gfCNCPoint1[18036] = {X 7.8608, Y 36.7035, Z -1.3333, A 0.000, B 0.000, C 0.000 }
gfCNCPoint1[18037] = {X 8.3776, Y 37.1520, Z -1.3333, A 0.000, B 0.000, C 0.000 }
gfCNCPoint1[18038] = {X 9.1826, Y 37.5595, Z -1.3333, A 0.000, B 0.000, C 0.000 }
gfCNCPoint1[18039] = {X 10.0390, Y 37.8436, Z -1.3333, A 0.000, B 0.000, C 0.000 }
gfCNCPoint1[18040] = {X 11.3458, Y 38.0858, Z -1.3333, A 0.000, B 0.000, C 0.000 }
gfCNCPoint1[18041] = {X 12.6726, Y 38.1626, Z -1.3333, A 0.000, B 0.000, C 0.000 }
gfCNCPoint1[18042] = {X 13.9985, Y 38.0726, Z -1.3333, A 0.000, B 0.000, C 0.000 }
gfCNCPoint1[18043] = {X 15.3028, Y 37.8174, Z -1.3333, A 0.000, B 0.000, C 0.000 }
gfCNCPoint1[18044] = {X 16.5649, Y 37.4009, Z -1.3333, A 0.000, B 0.000, C 0.000 }
gfCNCPoint1[18045] = {X 17.9591, Y 36.7477, Z -1.3333, A 0.000, B 0.000, C 0.000 }
gfCNCPoint1[18046] = {X 19.2706, Y 35.9412, Z -1.3333, A 0.000, B 0.000, C 0.000 }
gfCNCPoint1[18047] = {X 19.3492, Y 35.2028, Z -1.3333, A 0.000, B 0.000, C 0.000 }
gfCNCPoint1[18048] = {X 19.5579, Y 34.4902, Z -1.3333, A 0.000, B 0.000, C 0.000 }
gfCNCPoint1[18049] = {X 19.8900, Y 33.8261, Z -1.3333, A 0.000, B 0.000, C 0.000 }
gfCNCPoint1[18050] = {X 18.0017, Y 34.1716, Z -1.3333, A 0.000, B 0.000, C 0.000 }
gfCNCPoint1[18051] = {X 16.0932, Y 34.3789, Z -1.3333, A 0.000, B 0.000, C 0.000 }
gfCNCPoint1[18052] = {X 15.3691, Y 34.4315, Z -1.3333, A 0.000, B 0.000, C 0.000 }
gfCNCPoint1[18053] = {X 14.6448, Y 34.4821, Z -1.3333, A 0.000, B 0.000, C 0.000 }
gfCNCPoint1[18054] = {X 10.6931, Y 35.1018, Z -1.3333, A 0.000, B 0.000, C 0.000 }
gfCNCPoint1[18055] = {X 18.6386, Y 34.4782, Z -1.3333, A 0.000, B 0.000, C 0.000 }
gfCNCPoint1[18056] = {X 14.6393, Y 34.4023, Z -1.3333, A 0.000, B 0.000, C 0.000 }
gfCNCPoint1[18057] = {X 12.2464, Y 34.5545, Z -1.3333, A 0.000, B 0.000, C 0.000 }
gfCNCPoint1[18058] = {X 9.8522, Y 34.6839, Z -1.3333, A 0.000, B 0.000, C 0.000 }
gfCNCPoint1[18059] = {X 8.6234, Y 34.7897, Z -1.3333, A 0.000, B 0.000, C 0.000 }
gfCNCPoint1[18060] = {X 7.4164, Y 35.0431, Z -1.3333, A 0.000, B 0.000, C 0.000 }
gfCNCPoint1[18061] = {X 7.3529, Y 35.2331, Z -1.3333, A 0.000, B 0.000, C 0.000 }
gfCNCPoint1[18062] = {X 7.3309, Y 35.4323, Z -1.3333, A 0.000, B 0.000, C 0.000 }
gfCNCPoint1[18063] = {X 7.3977, Y 35.9629, Z -1.3333, A 0.000, B 0.000, C 0.000 }
gfCNCPoint1[18064] = {X 7.5977, Y 36.4590, Z -1.3333, A 0.000, B 0.000, C 0.000 }
gfCNCPoint1[18065] = {X 7.9176, Y 36.8876, Z -1.3333, A 0.000, B 0.000, C 0.000 }
gfCNCPoint1[18066] = {X 8.3362, Y 37.2205, Z -1.3333, A 0.000, B 0.000, C 0.000 }
gfCNCPoint1[18067] = {X 9.1519, Y 37.6334, Z -1.3333, A 0.000, B 0.000, C 0.000 }
gfCNCPoint1[18068] = {X 10.0195, Y 37.9212, Z -1.3333, A 0.000, B 0.000, C 0.000 }
gfCNCPoint1[18069] = {X 11.3362, Y 38.1652, Z -1.3333, A 0.000, B 0.000, C 0.000 }
gfCNCPoint1[18070] = {X 12.6730, Y 38.2425, Z -1.3333, A 0.000, B 0.000, C 0.000 }
gfCNCPoint1[18071] = {X 14.0089, Y 38.1519, Z -1.3333, A 0.000, B 0.000, C 0.000 }
gfCNCPoint1[18072] = {X 15.3231, Y 37.8948, Z -1.3333, A 0.000, B 0.000, C 0.000 }
gfCNCPoint1[18073] = {X 16.5947, Y 37.4752, Z -1.3333, A 0.000, B 0.000, C 0.000 }
gfCNCPoint1[18074] = {X 18.0152, Y 36.8083, Z -1.3333, A 0.000, B 0.000, C 0.000 }
gfCNCPoint1[18075] = {X 19.3501, Y 35.9832, Z -1.3333, A 0.000, B 0.000, C 0.000 }
gfCNCPoint1[18076] = {X 19.4352, Y 35.1814, Z -1.3333, A 0.000, B 0.000, C 0.000 }
gfCNCPoint1[18077] = {X 19.6764, Y 34.4119, Z -1.3333, A 0.000, B 0.000, C 0.000 }
gfCNCPoint1[18078] = {X 20.0642, Y 33.7049, Z -1.3333, A 0.000, B 0.000, C 0.000 }
gfCNCPoint1[18079] = {X 18.0872, Y 34.0781, Z -1.3333, A 0.000, B 0.000, C 0.000 }
gfCNCPoint1[18080] = {X 16.0874, Y 34.2991, Z -1.3333, A 0.000, B 0.000, C 0.000 }
gfCNCPoint1[18081] = {X 15.3634, Y 34.3517, Z -1.3333, A 0.000, B 0.000, C 0.000 }
gfCNCPoint1[18082] = {X 14.6393, Y 34.4023, Z -1.3333, A 0.000, B 0.000, C 0.000 }
gfCNCPoint1[18083] = {X 10.6876, Y 35.0220, Z -1.3333, A 0.000, B 0.000, C 0.000 }
gfCNCPoint1[18084] = {X 14.7703, Y 36.3178, Z -1.3333, A 0.000, B 0.000, C 0.000 }
gfCNCPoint1[18085] = {X 14.6338, Y 34.3225, Z -1.3333, A 0.000, B 0.000, C 0.000 }
gfCNCPoint1[18086] = {X 12.2422, Y 34.4746, Z -1.3333, A 0.000, B 0.000, C 0.000 }
gfCNCPoint1[18087] = {X 9.8492, Y 34.6040, Z -1.3333, A 0.000, B 0.000, C 0.000 }
gfCNCPoint1[18088] = {X 8.5932, Y 34.7133, Z -1.3333, A 0.000, B 0.000, C 0.000 }
gfCNCPoint1[18089] = {X 7.3600, Y 34.9757, Z -1.3333, A 0.000, B 0.000, C 0.000 }
gfCNCPoint1[18090] = {X 7.2790, Y 35.1975, Z -1.3333, A 0.000, B 0.000, C 0.000 }
gfCNCPoint1[18091] = {X 7.2509, Y 35.4320, Z -1.3333, A 0.000, B 0.000, C 0.000 }
gfCNCPoint1[18092] = {X 7.3203, Y 35.9830, Z -1.3333, A 0.000, B 0.000, C 0.000 }
gfCNCPoint1[18093] = {X 7.5280, Y 36.4982, Z -1.3333, A 0.000, B 0.000, C 0.000 }
gfCNCPoint1[18094] = {X 7.8602, Y 36.9433, Z -1.3333, A 0.000, B 0.000, C 0.000 }
gfCNCPoint1[18095] = {X 8.2949, Y 37.2890, Z -1.3333, A 0.000, B 0.000, C 0.000 }
gfCNCPoint1[18096] = {X 9.1211, Y 37.7073, Z -1.3333, A 0.000, B 0.000, C 0.000 }
gfCNCPoint1[18097] = {X 10.0001, Y 37.9988, Z -1.3333, A 0.000, B 0.000, C 0.000 }
gfCNCPoint1[18098] = {X 11.3265, Y 38.2446, Z -1.3333, A 0.000, B 0.000, C 0.000 }
gfCNCPoint1[18099] = {X 12.6734, Y 38.3225, Z -1.3333, A 0.000, B 0.000, C 0.000 }
gfCNCPoint1[18100] = {X 14.0194, Y 38.2312, Z -1.3333, A 0.000, B 0.000, C 0.000 }
gfCNCPoint1[18101] = {X 15.3433, Y 37.9722, Z -1.3333, A 0.000, B 0.000, C 0.000 }
gfCNCPoint1[18102] = {X 16.6244, Y 37.5494, Z -1.3333, A 0.000, B 0.000, C 0.000 }
gfCNCPoint1[18103] = {X 18.0716, Y 36.8688, Z -1.3333, A 0.000, B 0.000, C 0.000 }
gfCNCPoint1[18104] = {X 19.4300, Y 36.0248, Z -1.3333, A 0.000, B 0.000, C 0.000 }
gfCNCPoint1[18105] = {X 19.5226, Y 35.1553, Z -1.3333, A 0.000, B 0.000, C 0.000 }
gfCNCPoint1[18106] = {X 19.8019, Y 34.3266, Z -1.3333, A 0.000, B 0.000, C 0.000 }
gfCNCPoint1[18107] = {X 20.2547, Y 33.5784, Z -1.3333, A 0.000, B 0.000, C 0.000 }
gfCNCPoint1[18108] = {X 18.1810, Y 33.9830, Z -1.3333, A 0.000, B 0.000, C 0.000 }
gfCNCPoint1[18109] = {X 16.0816, Y 34.2193, Z -1.3333, A 0.000, B 0.000, C 0.000 }
gfCNCPoint1[18110] = {X 15.3578, Y 34.2719, Z -1.3333, A 0.000, B 0.000, C 0.000 }
gfCNCPoint1[18111] = {X 14.6338, Y 34.3225, Z -1.3333, A 0.000, B 0.000, C 0.000 }
gfCNCPoint1[18112] = {X 14.7703, Y 36.3178, Z -1.3333, A 0.000, B 0.000, C 0.000 }
gfCNCPoint1[18113] = {X 14.7703, Y 36.3178, Z 1.6667, A 0.000, B 0.000, C 0.000 }
gfCNCPoint1[18114] = {X 14.7703, Y 36.3178, Z 11.0000, A 0.000, B 0.000, C 0.000 }
gfCNCPoint1[18115] = {X 15.0706, Y 19.4899, Z 11.0000, A 0.000, B 0.000, C 0.000 }
gfCNCPoint1[18116] = {X 15.0706, Y 19.4899, Z 2.5000, A 0.000, B 0.000, C 0.000 }
gfCNCPoint1[18117] = {X 14.5039, Y 19.3617, Z 2.3443, A 0.000, B 0.000, C 0.000 }
gfCNCPoint1[18118] = {X 13.3045, Y 19.2481, Z 2.0215, A 0.000, B 0.000, C 0.000 }
gfCNCPoint1[18119] = {X 12.0998, Y 19.2655, Z 1.6987, A 0.000, B 0.000, C 0.000 }
gfCNCPoint1[18120] = {X 11.2937, Y 19.3811, Z 1.4805, A 0.000, B 0.000, C 0.000 }
gfCNCPoint1[18121] = {X 10.6070, Y 19.4891, Z 1.2942, A 0.000, B 0.000, C 0.000 }
gfCNCPoint1[18122] = {X 9.8986, Y 19.6124, Z 1.1015, A 0.000, B 0.000, C 0.000 }
gfCNCPoint1[18123] = {X 8.6156, Y 20.0582, Z 0.7376, A 0.000, B 0.000, C 0.000 }
gfCNCPoint1[18124] = {X 7.9834, Y 20.4007, Z 0.5449, A 0.000, B 0.000, C 0.000 }
gfCNCPoint1[18125] = {X 7.9275, Y 20.9124, Z 0.4070, A 0.000, B 0.000, C 0.000 }
gfCNCPoint1[18126] = {X 7.4464, Y 22.1372, Z 0.0544, A 0.000, B 0.000, C 0.000 }
gfCNCPoint1[18127] = {X 7.1391, Y 22.5500, Z -0.0835, A 0.000, B 0.000, C 0.000 }
gfCNCPoint1[18128] = {X 8.7346, Y 22.3449, Z -0.5145, A 0.000, B 0.000, C 0.000 }
gfCNCPoint1[18129] = {X 9.6130, Y 22.2741, Z -0.7506, A 0.000, B 0.000, C 0.000 }
gfCNCPoint1[18130] = {X 11.2207, Y 22.2213, Z -1.1817, A 0.000, B 0.000, C 0.000 }
gfCNCPoint1[18131] = {X 11.5036, Y 22.2116, Z -1.2575, A 0.000, B 0.000, C 0.000 }
gfCNCPoint1[18132] = {X 11.7864, Y 22.2003, Z -1.3333, A 0.000, B 0.000, C 0.000 }
gfCNCPoint1[18133] = {X 14.1145, Y 22.0807, Z -1.3333, A 0.000, B 0.000, C 0.000 }
gfCNCPoint1[18134] = {X 16.4392, Y 21.9079, Z -1.3333, A 0.000, B 0.000, C 0.000 }
gfCNCPoint1[18135] = {X 17.0540, Y 21.8327, Z -1.3333, A 0.000, B 0.000, C 0.000 }
gfCNCPoint1[18136] = {X 17.6536, Y 21.6779, Z -1.3333, A 0.000, B 0.000, C 0.000 }
gfCNCPoint1[18137] = {X 17.6759, Y 21.2173, Z -1.3333, A 0.000, B 0.000, C 0.000 }
gfCNCPoint1[18138] = {X 17.5258, Y 20.7814, Z -1.3333, A 0.000, B 0.000, C 0.000 }
gfCNCPoint1[18139] = {X 17.2248, Y 20.4321, Z -1.3333, A 0.000, B 0.000, C 0.000 }
gfCNCPoint1[18140] = {X 16.3055, Y 19.8916, Z -1.3333, A 0.000, B 0.000, C 0.000 }
gfCNCPoint1[18141] = {X 15.2982, Y 19.5414, Z -1.3333, A 0.000, B 0.000, C 0.000 }
gfCNCPoint1[18142] = {X 13.9732, Y 19.3253, Z -1.3333, A 0.000, B 0.000, C 0.000 }
gfCNCPoint1[18143] = {X 12.6317, Y 19.2716, Z -1.3333, A 0.000, B 0.000, C 0.000 }
gfCNCPoint1[18144] = {X 11.2937, Y 19.3811, Z -1.3333, A 0.000, B 0.000, C 0.000 }
gfCNCPoint1[18145] = {X 10.6070, Y 19.4891, Z -1.3333, A 0.000, B 0.000, C 0.000 }
gfCNCPoint1[18146] = {X 9.2582, Y 19.8383, Z -1.3333, A 0.000, B 0.000, C 0.000 }
gfCNCPoint1[18147] = {X 7.9834, Y 20.4007, Z -1.3333, A 0.000, B 0.000, C 0.000 }
gfCNCPoint1[18148] = {X 7.8310, Y 21.1635, Z -1.3333, A 0.000, B 0.000, C 0.000 }
gfCNCPoint1[18149] = {X 7.5466, Y 21.8875, Z -1.3333, A 0.000, B 0.000, C 0.000 }
gfCNCPoint1[18150] = {X 7.1391, Y 22.5500, Z -1.3333, A 0.000, B 0.000, C 0.000 }
gfCNCPoint1[18151] = {X 9.1760, Y 22.3372, Z -1.3333, A 0.000, B 0.000, C 0.000 }
gfCNCPoint1[18152] = {X 11.2207, Y 22.2213, Z -1.3333, A 0.000, B 0.000, C 0.000 }
gfCNCPoint1[18153] = {X 11.5036, Y 22.2112, Z -1.3333, A 0.000, B 0.000, C 0.000 }
gfCNCPoint1[18154] = {X 11.7864, Y 22.2003, Z -1.3333, A 0.000, B 0.000, C 0.000 }
gfCNCPoint1[18155] = {X 7.7941, Y 22.0908, Z -1.3333, A 0.000, B 0.000, C 0.000 }
gfCNCPoint1[18156] = {X 11.7896, Y 22.2802, Z -1.3333, A 0.000, B 0.000, C 0.000 }
gfCNCPoint1[18157] = {X 14.1160, Y 22.1607, Z -1.3333, A 0.000, B 0.000, C 0.000 }
gfCNCPoint1[18158] = {X 16.4391, Y 21.9880, Z -1.3333, A 0.000, B 0.000, C 0.000 }
gfCNCPoint1[18159] = {X 17.0880, Y 21.9077, Z -1.3333, A 0.000, B 0.000, C 0.000 }
gfCNCPoint1[18160] = {X 17.7200, Y 21.7400, Z -1.3333, A 0.000, B 0.000, C 0.000 }
gfCNCPoint1[18161] = {X 17.7589, Y 21.2351, Z -1.3333, A 0.000, B 0.000, C 0.000 }
gfCNCPoint1[18162] = {X 17.6020, Y 20.7536, Z -1.3333, A 0.000, B 0.000, C 0.000 }
gfCNCPoint1[18163] = {X 17.2732, Y 20.3684, Z -1.3333, A 0.000, B 0.000, C 0.000 }
gfCNCPoint1[18164] = {X 16.3395, Y 19.8192, Z -1.3333, A 0.000, B 0.000, C 0.000 }
gfCNCPoint1[18165] = {X 15.3164, Y 19.4635, Z -1.3333, A 0.000, B 0.000, C 0.000 }
gfCNCPoint1[18166] = {X 13.9814, Y 19.2457, Z -1.3333, A 0.000, B 0.000, C 0.000 }
gfCNCPoint1[18167] = {X 12.6299, Y 19.1916, Z -1.3333, A 0.000, B 0.000, C 0.000 }
gfCNCPoint1[18168] = {X 11.2818, Y 19.3020, Z -1.3333, A 0.000, B 0.000, C 0.000 }
gfCNCPoint1[18169] = {X 10.5939, Y 19.4102, Z -1.3333, A 0.000, B 0.000, C 0.000 }
gfCNCPoint1[18170] = {X 9.2123, Y 19.7696, Z -1.3333, A 0.000, B 0.000, C 0.000 }
gfCNCPoint1[18171] = {X 7.9082, Y 20.3506, Z -1.3333, A 0.000, B 0.000, C 0.000 }
gfCNCPoint1[18172] = {X 7.7437, Y 21.1760, Z -1.3333, A 0.000, B 0.000, C 0.000 }
gfCNCPoint1[18173] = {X 7.4223, Y 21.9539, Z -1.3333, A 0.000, B 0.000, C 0.000 }
gfCNCPoint1[18174] = {X 6.9562, Y 22.6547, Z -1.3333, A 0.000, B 0.000, C 0.000 }
gfCNCPoint1[18175] = {X 9.0854, Y 22.4248, Z -1.3333, A 0.000, B 0.000, C 0.000 }
gfCNCPoint1[18176] = {X 11.2234, Y 22.3012, Z -1.3333, A 0.000, B 0.000, C 0.000 }
gfCNCPoint1[18177] = {X 11.5065, Y 22.2911, Z -1.3333, A 0.000, B 0.000, C 0.000 }
gfCNCPoint1[18178] = {X 11.7896, Y 22.2802, Z -1.3333, A 0.000, B 0.000, C 0.000 }
gfCNCPoint1[18179] = {X 15.7573, Y 21.7730, Z -1.3333, A 0.000, B 0.000, C 0.000 }
gfCNCPoint1[18180] = {X 7.7973, Y 22.1707, Z -1.3333, A 0.000, B 0.000, C 0.000 }
gfCNCPoint1[18181] = {X 11.7928, Y 22.3601, Z -1.3333, A 0.000, B 0.000, C 0.000 }
gfCNCPoint1[18182] = {X 14.1204, Y 22.2406, Z -1.3333, A 0.000, B 0.000, C 0.000 }
gfCNCPoint1[18183] = {X 16.4447, Y 22.0679, Z -1.3333, A 0.000, B 0.000, C 0.000 }
gfCNCPoint1[18184] = {X 17.1242, Y 21.9821, Z -1.3333, A 0.000, B 0.000, C 0.000 }
gfCNCPoint1[18185] = {X 17.7850, Y 21.8022, Z -1.3333, A 0.000, B 0.000, C 0.000 }
gfCNCPoint1[18186] = {X 17.8413, Y 21.2532, Z -1.3333, A 0.000, B 0.000, C 0.000 }
gfCNCPoint1[18187] = {X 17.6781, Y 20.7259, Z -1.3333, A 0.000, B 0.000, C 0.000 }
gfCNCPoint1[18188] = {X 17.3216, Y 20.3046, Z -1.3333, A 0.000, B 0.000, C 0.000 }
gfCNCPoint1[18189] = {X 16.3735, Y 19.7468, Z -1.3333, A 0.000, B 0.000, C 0.000 }
gfCNCPoint1[18190] = {X 15.3345, Y 19.3856, Z -1.3333, A 0.000, B 0.000, C 0.000 }
gfCNCPoint1[18191] = {X 13.9896, Y 19.1661, Z -1.3333, A 0.000, B 0.000, C 0.000 }
gfCNCPoint1[18192] = {X 12.6280, Y 19.1116, Z -1.3333, A 0.000, B 0.000, C 0.000 }
gfCNCPoint1[18193] = {X 11.2699, Y 19.2229, Z -1.3333, A 0.000, B 0.000, C 0.000 }
gfCNCPoint1[18194] = {X 10.5809, Y 19.3312, Z -1.3333, A 0.000, B 0.000, C 0.000 }
gfCNCPoint1[18195] = {X 9.6302, Y 19.5517, Z -1.3333, A 0.000, B 0.000, C 0.000 }
gfCNCPoint1[18196] = {X 8.7100, Y 19.8764, Z -1.3333, A 0.000, B 0.000, C 0.000 }
gfCNCPoint1[18197] = {X 7.8316, Y 20.3015, Z -1.3333, A 0.000, B 0.000, C 0.000 }
gfCNCPoint1[18198] = {X 7.8286, Y 20.3427, Z -1.3333, A 0.000, B 0.000, C 0.000 }
gfCNCPoint1[18199] = {X 7.6465, Y 21.2191, Z -1.3333, A 0.000, B 0.000, C 0.000 }
gfCNCPoint1[18200] = {X 7.2844, Y 22.0378, Z -1.3333, A 0.000, B 0.000, C 0.000 }
gfCNCPoint1[18201] = {X 6.7585, Y 22.7622, Z -1.3333, A 0.000, B 0.000, C 0.000 }
gfCNCPoint1[18202] = {X 8.9873, Y 22.5134, Z -1.3333, A 0.000, B 0.000, C 0.000 }
gfCNCPoint1[18203] = {X 11.2261, Y 22.3812, Z -1.3333, A 0.000, B 0.000, C 0.000 }
gfCNCPoint1[18204] = {X 11.5095, Y 22.3711, Z -1.3333, A 0.000, B 0.000, C 0.000 }
gfCNCPoint1[18205] = {X 11.7928, Y 22.3601, Z -1.3333, A 0.000, B 0.000, C 0.000 }
gfCNCPoint1[18206] = {X 15.7605, Y 21.8529, Z -1.3333, A 0.000, B 0.000, C 0.000 }
gfCNCPoint1[18207] = {X 7.8005, Y 22.2506, Z -1.3333, A 0.000, B 0.000, C 0.000 }
gfCNCPoint1[18208] = {X 11.7960, Y 22.4401, Z -1.3333, A 0.000, B 0.000, C 0.000 }
gfCNCPoint1[18209] = {X 14.1248, Y 22.3205, Z -1.3333, A 0.000, B 0.000, C 0.000 }
gfCNCPoint1[18210] = {X 16.4504, Y 22.1477, Z -1.3333, A 0.000, B 0.000, C 0.000 }
gfCNCPoint1[18211] = {X 17.1598, Y 22.0566, Z -1.3333, A 0.000, B 0.000, C 0.000 }
gfCNCPoint1[18212] = {X 17.8488, Y 21.8646, Z -1.3333, A 0.000, B 0.000, C 0.000 }
gfCNCPoint1[18213] = {X 17.9277, Y 21.4220, Z -1.3333, A 0.000, B 0.000, C 0.000 }
gfCNCPoint1[18214] = {X 17.8684, Y 20.9763, Z -1.3333, A 0.000, B 0.000, C 0.000 }
gfCNCPoint1[18215] = {X 17.6764, Y 20.5698, Z -1.3333, A 0.000, B 0.000, C 0.000 }
gfCNCPoint1[18216] = {X 17.3699, Y 20.2409, Z -1.3333, A 0.000, B 0.000, C 0.000 }
gfCNCPoint1[18217] = {X 16.4075, Y 19.6744, Z -1.3333, A 0.000, B 0.000, C 0.000 }
gfCNCPoint1[18218] = {X 15.3527, Y 19.3077, Z -1.3333, A 0.000, B 0.000, C 0.000 }
gfCNCPoint1[18219] = {X 13.9979, Y 19.0866, Z -1.3333, A 0.000, B 0.000, C 0.000 }
gfCNCPoint1[18220] = {X 12.6262, Y 19.0317, Z -1.3333, A 0.000, B 0.000, C 0.000 }
gfCNCPoint1[18221] = {X 11.2580, Y 19.1438, Z -1.3333, A 0.000, B 0.000, C 0.000 }
gfCNCPoint1[18222] = {X 10.5678, Y 19.2523, Z -1.3333, A 0.000, B 0.000, C 0.000 }
gfCNCPoint1[18223] = {X 9.5943, Y 19.4788, Z -1.3333, A 0.000, B 0.000, C 0.000 }
gfCNCPoint1[18224] = {X 8.6526, Y 19.8137, Z -1.3333, A 0.000, B 0.000, C 0.000 }
gfCNCPoint1[18225] = {X 7.7547, Y 20.2528, Z -1.3333, A 0.000, B 0.000, C 0.000 }
gfCNCPoint1[18226] = {X 7.7493, Y 20.3317, Z -1.3333, A 0.000, B 0.000, C 0.000 }
gfCNCPoint1[18227] = {X 7.5471, Y 21.2648, Z -1.3333, A 0.000, B 0.000, C 0.000 }
gfCNCPoint1[18228] = {X 7.1375, Y 22.1272, Z -1.3333, A 0.000, B 0.000, C 0.000 }
gfCNCPoint1[18229] = {X 6.5421, Y 22.8735, Z -1.3333, A 0.000, B 0.000, C 0.000 }
gfCNCPoint1[18230] = {X 8.8798, Y 22.6030, Z -1.3333, A 0.000, B 0.000, C 0.000 }
gfCNCPoint1[18231] = {X 11.2288, Y 22.4611, Z -1.3333, A 0.000, B 0.000, C 0.000 }
gfCNCPoint1[18232] = {X 11.5124, Y 22.4510, Z -1.3333, A 0.000, B 0.000, C 0.000 }
gfCNCPoint1[18233] = {X 11.7960, Y 22.4401, Z -1.3333, A 0.000, B 0.000, C 0.000 }
gfCNCPoint1[18234] = {X 15.7637, Y 21.9328, Z -1.3333, A 0.000, B 0.000, C 0.000 }
gfCNCPoint1[18235] = {X 7.8037, Y 22.3306, Z -1.3333, A 0.000, B 0.000, C 0.000 }
gfCNCPoint1[18236] = {X 11.7992, Y 22.5200, Z -1.3333, A 0.000, B 0.000, C 0.000 }
gfCNCPoint1[18237] = {X 14.1293, Y 22.4004, Z -1.3333, A 0.000, B 0.000, C 0.000 }
gfCNCPoint1[18238] = {X 16.4560, Y 22.2275, Z -1.3333, A 0.000, B 0.000, C 0.000 }
gfCNCPoint1[18239] = {X 17.1948, Y 22.1310, Z -1.3333, A 0.000, B 0.000, C 0.000 }
gfCNCPoint1[18240] = {X 17.9114, Y 21.9269, Z -1.3333, A 0.000, B 0.000, C 0.000 }
gfCNCPoint1[18241] = {X 18.0068, Y 21.4523, Z -1.3333, A 0.000, B 0.000, C 0.000 }
gfCNCPoint1[18242] = {X 17.9503, Y 20.9716, Z -1.3333, A 0.000, B 0.000, C 0.000 }
gfCNCPoint1[18243] = {X 17.7474, Y 20.5320, Z -1.3333, A 0.000, B 0.000, C 0.000 }
gfCNCPoint1[18244] = {X 17.4182, Y 20.1771, Z -1.3333, A 0.000, B 0.000, C 0.000 }
gfCNCPoint1[18245] = {X 16.4415, Y 19.6020, Z -1.3333, A 0.000, B 0.000, C 0.000 }
gfCNCPoint1[18246] = {X 15.3709, Y 19.2298, Z -1.3333, A 0.000, B 0.000, C 0.000 }
gfCNCPoint1[18247] = {X 14.0061, Y 19.0070, Z -1.3333, A 0.000, B 0.000, C 0.000 }
gfCNCPoint1[18248] = {X 12.6243, Y 18.9517, Z -1.3333, A 0.000, B 0.000, C 0.000 }
gfCNCPoint1[18249] = {X 11.2461, Y 19.0647, Z -1.3333, A 0.000, B 0.000, C 0.000 }
gfCNCPoint1[18250] = {X 10.5548, Y 19.1734, Z -1.3333, A 0.000, B 0.000, C 0.000 }
gfCNCPoint1[18251] = {X 9.5584, Y 19.4060, Z -1.3333, A 0.000, B 0.000, C 0.000 }
gfCNCPoint1[18252] = {X 8.5952, Y 19.7511, Z -1.3333, A 0.000, B 0.000, C 0.000 }
gfCNCPoint1[18253] = {X 7.6779, Y 20.2043, Z -1.3333, A 0.000, B 0.000, C 0.000 }
gfCNCPoint1[18254] = {X 7.6696, Y 20.3250, Z -1.3333, A 0.000, B 0.000, C 0.000 }
gfCNCPoint1[18255] = {X 7.5229, Y 21.0766, Z -1.3333, A 0.000, B 0.000, C 0.000 }
gfCNCPoint1[18256] = {X 7.2384, Y 21.7876, Z -1.3333, A 0.000, B 0.000, C 0.000 }
gfCNCPoint1[18257] = {X 6.8261, Y 22.4329, Z -1.3333, A 0.000, B 0.000, C 0.000 }
gfCNCPoint1[18258] = {X 6.3004, Y 22.9898, Z -1.3333, A 0.000, B 0.000, C 0.000 }
gfCNCPoint1[18259] = {X 8.7595, Y 22.6941, Z -1.3333, A 0.000, B 0.000, C 0.000 }
gfCNCPoint1[18260] = {X 11.2315, Y 22.5411, Z -1.3333, A 0.000, B 0.000, C 0.000 }
gfCNCPoint1[18261] = {X 11.5153, Y 22.5310, Z -1.3333, A 0.000, B 0.000, C 0.000 }
gfCNCPoint1[18262] = {X 11.7992, Y 22.5200, Z -1.3333, A 0.000, B 0.000, C 0.000 }
gfCNCPoint1[18263] = {X 15.7669, Y 22.0128, Z -1.3333, A 0.000, B 0.000, C 0.000 }
gfCNCPoint1[18264] = {X 11.7273, Y 22.6029, Z -1.3333, A 0.000, B 0.000, C 0.000 }
gfCNCPoint1[18265] = {X 11.8024, Y 22.6000, Z -1.3333, A 0.000, B 0.000, C 0.000 }
gfCNCPoint1[18266] = {X 14.1337, Y 22.4802, Z -1.3333, A 0.000, B 0.000, C 0.000 }
gfCNCPoint1[18267] = {X 16.4617, Y 22.3073, Z -1.3333, A 0.000, B 0.000, C 0.000 }
gfCNCPoint1[18268] = {X 17.2294, Y 22.2056, Z -1.3333, A 0.000, B 0.000, C 0.000 }
gfCNCPoint1[18269] = {X 17.9731, Y 21.9894, Z -1.3333, A 0.000, B 0.000, C 0.000 }
gfCNCPoint1[18270] = {X 18.0854, Y 21.4830, Z -1.3333, A 0.000, B 0.000, C 0.000 }
gfCNCPoint1[18271] = {X 18.0320, Y 20.9671, Z -1.3333, A 0.000, B 0.000, C 0.000 }
gfCNCPoint1[18272] = {X 17.8185, Y 20.4944, Z -1.3333, A 0.000, B 0.000, C 0.000 }
gfCNCPoint1[18273] = {X 17.4665, Y 20.1133, Z -1.3333, A 0.000, B 0.000, C 0.000 }
gfCNCPoint1[18274] = {X 16.4755, Y 19.5295, Z -1.3333, A 0.000, B 0.000, C 0.000 }
gfCNCPoint1[18275] = {X 15.3891, Y 19.1519, Z -1.3333, A 0.000, B 0.000, C 0.000 }
gfCNCPoint1[18276] = {X 14.0143, Y 18.9274, Z -1.3333, A 0.000, B 0.000, C 0.000 }
gfCNCPoint1[18277] = {X 12.6225, Y 18.8717, Z -1.3333, A 0.000, B 0.000, C 0.000 }
gfCNCPoint1[18278] = {X 11.2342, Y 18.9856, Z -1.3333, A 0.000, B 0.000, C 0.000 }
gfCNCPoint1[18279] = {X 10.5417, Y 19.0944, Z -1.3333, A 0.000, B 0.000, C 0.000 }
gfCNCPoint1[18280] = {X 9.5224, Y 19.3332, Z -1.3333, A 0.000, B 0.000, C 0.000 }
gfCNCPoint1[18281] = {X 8.5377, Y 19.6887, Z -1.3333, A 0.000, B 0.000, C 0.000 }
gfCNCPoint1[18282] = {X 7.6010, Y 20.1561, Z -1.3333, A 0.000, B 0.000, C 0.000 }
gfCNCPoint1[18283] = {X 7.5898, Y 20.3183, Z -1.3333, A 0.000, B 0.000, C 0.000 }
gfCNCPoint1[18284] = {X 7.4460, Y 21.0549, Z -1.3333, A 0.000, B 0.000, C 0.000 }
gfCNCPoint1[18285] = {X 7.1670, Y 21.7516, Z -1.3333, A 0.000, B 0.000, C 0.000 }
gfCNCPoint1[18286] = {X 6.7628, Y 22.3840, Z -1.3333, A 0.000, B 0.000, C 0.000 }
gfCNCPoint1[18287] = {X 6.2476, Y 22.9297, Z -1.3333, A 0.000, B 0.000, C 0.000 }
gfCNCPoint1[18288] = {X 6.2069, Y 22.9649, Z -1.3333, A 0.000, B 0.000, C 0.000 }
gfCNCPoint1[18289] = {X 6.1658, Y 22.9996, Z -1.3333, A 0.000, B 0.000, C 0.000 }
gfCNCPoint1[18290] = {X 6.1504, Y 23.0935, Z -1.3333, A 0.000, B 0.000, C 0.000 }
gfCNCPoint1[18291] = {X 6.2313, Y 23.0811, Z -1.3333, A 0.000, B 0.000, C 0.000 }
gfCNCPoint1[18292] = {X 6.3123, Y 23.0689, Z -1.3333, A 0.000, B 0.000, C 0.000 }
gfCNCPoint1[18293] = {X 8.7667, Y 22.7737, Z -1.3333, A 0.000, B 0.000, C 0.000 }
gfCNCPoint1[18294] = {X 11.2342, Y 22.6210, Z -1.3333, A 0.000, B 0.000, C 0.000 }
gfCNCPoint1[18295] = {X 11.5183, Y 22.6109, Z -1.3333, A 0.000, B 0.000, C 0.000 }
gfCNCPoint1[18296] = {X 11.8024, Y 22.6000, Z -1.3333, A 0.000, B 0.000, C 0.000 }
gfCNCPoint1[18297] = {X 11.7226, Y 20.6015, Z -1.3333, A 0.000, B 0.000, C 0.000 }
gfCNCPoint1[18298] = {X 11.7226, Y 20.6015, Z 1.6667, A 0.000, B 0.000, C 0.000 }
gfCNCPoint1[18299] = {X 11.7226, Y 20.6015, Z 11.0000, A 0.000, B 0.000, C 0.000 }
gfCNCPoint1[18300] = {X 15.0739, Y 19.4910, Z 11.0000, A 0.000, B 0.000, C 0.000 }
gfCNCPoint1[18301] = {X 15.0739, Y 19.4910, Z 1.6667, A 0.000, B 0.000, C 0.000 }
gfCNCPoint1[18302] = {X 14.5039, Y 19.3620, Z 1.5101, A 0.000, B 0.000, C 0.000 }
gfCNCPoint1[18303] = {X 13.3045, Y 19.2484, Z 1.1873, A 0.000, B 0.000, C 0.000 }
gfCNCPoint1[18304] = {X 12.0998, Y 19.2658, Z 0.8644, A 0.000, B 0.000, C 0.000 }
gfCNCPoint1[18305] = {X 11.2937, Y 19.3815, Z 0.6462, A 0.000, B 0.000, C 0.000 }
gfCNCPoint1[18306] = {X 10.6070, Y 19.4894, Z 0.4600, A 0.000, B 0.000, C 0.000 }
gfCNCPoint1[18307] = {X 9.8987, Y 19.6126, Z 0.2673, A 0.000, B 0.000, C 0.000 }
gfCNCPoint1[18308] = {X 8.6154, Y 20.0585, Z -0.0967, A 0.000, B 0.000, C 0.000 }
gfCNCPoint1[18309] = {X 7.9834, Y 20.4011, Z -0.2893, A 0.000, B 0.000, C 0.000 }
gfCNCPoint1[18310] = {X 7.9275, Y 20.9127, Z -0.4272, A 0.000, B 0.000, C 0.000 }
gfCNCPoint1[18311] = {X 7.4486, Y 22.1334, Z -0.7786, A 0.000, B 0.000, C 0.000 }
gfCNCPoint1[18312] = {X 7.1417, Y 22.5465, Z -0.9165, A 0.000, B 0.000, C 0.000 }
gfCNCPoint1[18313] = {X 8.6586, Y 22.3495, Z -1.3263, A 0.000, B 0.000, C 0.000 }
gfCNCPoint1[18314] = {X 8.9966, Y 22.3205, Z -1.4172, A 0.000, B 0.000, C 0.000 }
gfCNCPoint1[18315] = {X 10.5268, Y 22.2562, Z -1.8276, A 0.000, B 0.000, C 0.000 }
gfCNCPoint1[18316] = {X 11.1590, Y 22.2325, Z -1.9971, A 0.000, B 0.000, C 0.000 }
gfCNCPoint1[18317] = {X 11.7911, Y 22.2034, Z -2.1667, A 0.000, B 0.000, C 0.000 }
gfCNCPoint1[18318] = {X 14.1196, Y 22.0775, Z -2.1667, A 0.000, B 0.000, C 0.000 }
gfCNCPoint1[18319] = {X 16.4458, Y 21.9144, Z -2.1667, A 0.000, B 0.000, C 0.000 }
gfCNCPoint1[18320] = {X 17.0568, Y 21.8305, Z -2.1667, A 0.000, B 0.000, C 0.000 }
gfCNCPoint1[18321] = {X 17.6538, Y 21.6758, Z -2.1667, A 0.000, B 0.000, C 0.000 }
gfCNCPoint1[18322] = {X 17.6753, Y 21.2161, Z -2.1667, A 0.000, B 0.000, C 0.000 }
gfCNCPoint1[18323] = {X 17.5252, Y 20.7810, Z -2.1667, A 0.000, B 0.000, C 0.000 }
gfCNCPoint1[18324] = {X 17.2248, Y 20.4324, Z -2.1667, A 0.000, B 0.000, C 0.000 }
gfCNCPoint1[18325] = {X 16.3055, Y 19.8919, Z -2.1667, A 0.000, B 0.000, C 0.000 }
gfCNCPoint1[18326] = {X 15.2982, Y 19.5418, Z -2.1667, A 0.000, B 0.000, C 0.000 }
gfCNCPoint1[18327] = {X 13.9732, Y 19.3256, Z -2.1667, A 0.000, B 0.000, C 0.000 }
gfCNCPoint1[18328] = {X 12.6317, Y 19.2719, Z -2.1667, A 0.000, B 0.000, C 0.000 }
gfCNCPoint1[18329] = {X 11.2937, Y 19.3815, Z -2.1667, A 0.000, B 0.000, C 0.000 }
gfCNCPoint1[18330] = {X 10.6070, Y 19.4894, Z -2.1667, A 0.000, B 0.000, C 0.000 }
gfCNCPoint1[18331] = {X 9.2581, Y 19.8386, Z -2.1667, A 0.000, B 0.000, C 0.000 }
gfCNCPoint1[18332] = {X 7.9834, Y 20.4011, Z -2.1667, A 0.000, B 0.000, C 0.000 }
gfCNCPoint1[18333] = {X 7.8313, Y 21.1623, Z -2.1667, A 0.000, B 0.000, C 0.000 }
gfCNCPoint1[18334] = {X 7.5478, Y 21.8850, Z -2.1667, A 0.000, B 0.000, C 0.000 }
gfCNCPoint1[18335] = {X 7.1417, Y 22.5465, Z -2.1667, A 0.000, B 0.000, C 0.000 }
gfCNCPoint1[18336] = {X 8.8311, Y 22.3645, Z -2.1667, A 0.000, B 0.000, C 0.000 }
gfCNCPoint1[18337] = {X 10.5268, Y 22.2562, Z -2.1667, A 0.000, B 0.000, C 0.000 }
gfCNCPoint1[18338] = {X 11.1590, Y 22.2311, Z -2.1667, A 0.000, B 0.000, C 0.000 }
gfCNCPoint1[18339] = {X 11.7911, Y 22.2034, Z -2.1667, A 0.000, B 0.000, C 0.000 }
gfCNCPoint1[18340] = {X 7.7982, Y 22.1185, Z -2.1667, A 0.000, B 0.000, C 0.000 }
gfCNCPoint1[18341] = {X 11.7948, Y 22.2833, Z -2.1667, A 0.000, B 0.000, C 0.000 }
gfCNCPoint1[18342] = {X 14.1246, Y 22.1573, Z -2.1667, A 0.000, B 0.000, C 0.000 }
gfCNCPoint1[18343] = {X 16.4521, Y 21.9941, Z -2.1667, A 0.000, B 0.000, C 0.000 }
gfCNCPoint1[18344] = {X 17.0939, Y 21.9046, Z -2.1667, A 0.000, B 0.000, C 0.000 }
gfCNCPoint1[18345] = {X 17.7202, Y 21.7382, Z -2.1667, A 0.000, B 0.000, C 0.000 }
gfCNCPoint1[18346] = {X 17.7584, Y 21.2340, Z -2.1667, A 0.000, B 0.000, C 0.000 }
gfCNCPoint1[18347] = {X 17.6015, Y 20.7533, Z -2.1667, A 0.000, B 0.000, C 0.000 }
gfCNCPoint1[18348] = {X 17.2732, Y 20.3687, Z -2.1667, A 0.000, B 0.000, C 0.000 }
gfCNCPoint1[18349] = {X 16.3395, Y 19.8195, Z -2.1667, A 0.000, B 0.000, C 0.000 }
gfCNCPoint1[18350] = {X 15.3164, Y 19.4639, Z -2.1667, A 0.000, B 0.000, C 0.000 }
gfCNCPoint1[18351] = {X 13.9814, Y 19.2461, Z -2.1667, A 0.000, B 0.000, C 0.000 }
gfCNCPoint1[18352] = {X 12.6299, Y 19.1919, Z -2.1667, A 0.000, B 0.000, C 0.000 }
gfCNCPoint1[18353] = {X 11.2818, Y 19.3024, Z -2.1667, A 0.000, B 0.000, C 0.000 }
gfCNCPoint1[18354] = {X 10.5939, Y 19.4105, Z -2.1667, A 0.000, B 0.000, C 0.000 }
gfCNCPoint1[18355] = {X 9.2122, Y 19.7699, Z -2.1667, A 0.000, B 0.000, C 0.000 }
gfCNCPoint1[18356] = {X 7.9082, Y 20.3510, Z -2.1667, A 0.000, B 0.000, C 0.000 }
gfCNCPoint1[18357] = {X 7.7440, Y 21.1749, Z -2.1667, A 0.000, B 0.000, C 0.000 }
gfCNCPoint1[18358] = {X 7.4235, Y 21.9516, Z -2.1667, A 0.000, B 0.000, C 0.000 }
gfCNCPoint1[18359] = {X 6.9588, Y 22.6515, Z -2.1667, A 0.000, B 0.000, C 0.000 }
gfCNCPoint1[18360] = {X 8.7399, Y 22.4527, Z -2.1667, A 0.000, B 0.000, C 0.000 }
gfCNCPoint1[18361] = {X 10.5283, Y 22.3362, Z -2.1667, A 0.000, B 0.000, C 0.000 }
gfCNCPoint1[18362] = {X 11.1616, Y 22.3111, Z -2.1667, A 0.000, B 0.000, C 0.000 }
gfCNCPoint1[18363] = {X 11.7948, Y 22.2833, Z -2.1667, A 0.000, B 0.000, C 0.000 }
gfCNCPoint1[18364] = {X 15.7593, Y 21.7516, Z -2.1667, A 0.000, B 0.000, C 0.000 }
gfCNCPoint1[18365] = {X 7.8018, Y 22.1984, Z -2.1667, A 0.000, B 0.000, C 0.000 }
gfCNCPoint1[18366] = {X 11.7984, Y 22.3632, Z -2.1667, A 0.000, B 0.000, C 0.000 }
gfCNCPoint1[18367] = {X 14.1295, Y 22.2371, Z -2.1667, A 0.000, B 0.000, C 0.000 }
gfCNCPoint1[18368] = {X 16.4583, Y 22.0739, Z -2.1667, A 0.000, B 0.000, C 0.000 }
gfCNCPoint1[18369] = {X 17.1303, Y 21.9789, Z -2.1667, A 0.000, B 0.000, C 0.000 }
gfCNCPoint1[18370] = {X 17.7851, Y 21.8008, Z -2.1667, A 0.000, B 0.000, C 0.000 }
gfCNCPoint1[18371] = {X 17.8409, Y 21.2524, Z -2.1667, A 0.000, B 0.000, C 0.000 }
gfCNCPoint1[18372] = {X 17.6777, Y 20.7258, Z -2.1667, A 0.000, B 0.000, C 0.000 }
gfCNCPoint1[18373] = {X 17.3216, Y 20.3049, Z -2.1667, A 0.000, B 0.000, C 0.000 }
gfCNCPoint1[18374] = {X 16.3735, Y 19.7471, Z -2.1667, A 0.000, B 0.000, C 0.000 }
gfCNCPoint1[18375] = {X 15.3346, Y 19.3860, Z -2.1667, A 0.000, B 0.000, C 0.000 }
gfCNCPoint1[18376] = {X 13.9896, Y 19.1665, Z -2.1667, A 0.000, B 0.000, C 0.000 }
gfCNCPoint1[18377] = {X 12.6280, Y 19.1120, Z -2.1667, A 0.000, B 0.000, C 0.000 }
gfCNCPoint1[18378] = {X 11.2699, Y 19.2233, Z -2.1667, A 0.000, B 0.000, C 0.000 }
gfCNCPoint1[18379] = {X 10.5809, Y 19.3316, Z -2.1667, A 0.000, B 0.000, C 0.000 }
gfCNCPoint1[18380] = {X 9.6302, Y 19.5519, Z -2.1667, A 0.000, B 0.000, C 0.000 }
gfCNCPoint1[18381] = {X 8.7100, Y 19.8767, Z -2.1667, A 0.000, B 0.000, C 0.000 }
gfCNCPoint1[18382] = {X 7.8316, Y 20.3018, Z -2.1667, A 0.000, B 0.000, C 0.000 }
gfCNCPoint1[18383] = {X 7.8286, Y 20.3430, Z -2.1667, A 0.000, B 0.000, C 0.000 }
gfCNCPoint1[18384] = {X 7.6468, Y 21.2182, Z -2.1667, A 0.000, B 0.000, C 0.000 }
gfCNCPoint1[18385] = {X 7.2856, Y 22.0358, Z -2.1667, A 0.000, B 0.000, C 0.000 }
gfCNCPoint1[18386] = {X 6.7610, Y 22.7595, Z -2.1667, A 0.000, B 0.000, C 0.000 }
gfCNCPoint1[18387] = {X 8.6421, Y 22.5418, Z -2.1667, A 0.000, B 0.000, C 0.000 }
gfCNCPoint1[18388] = {X 10.5316, Y 22.4161, Z -2.1667, A 0.000, B 0.000, C 0.000 }
gfCNCPoint1[18389] = {X 11.1651, Y 22.3910, Z -2.1667, A 0.000, B 0.000, C 0.000 }
gfCNCPoint1[18390] = {X 11.7984, Y 22.3632, Z -2.1667, A 0.000, B 0.000, C 0.000 }
gfCNCPoint1[18391] = {X 15.7629, Y 21.8315, Z -2.1667, A 0.000, B 0.000, C 0.000 }
gfCNCPoint1[18392] = {X 7.8055, Y 22.2783, Z -2.1667, A 0.000, B 0.000, C 0.000 }
gfCNCPoint1[18393] = {X 11.8021, Y 22.4431, Z -2.1667, A 0.000, B 0.000, C 0.000 }
gfCNCPoint1[18394] = {X 14.1345, Y 22.3170, Z -2.1667, A 0.000, B 0.000, C 0.000 }
gfCNCPoint1[18395] = {X 16.4645, Y 22.1536, Z -2.1667, A 0.000, B 0.000, C 0.000 }
gfCNCPoint1[18396] = {X 17.1660, Y 22.0532, Z -2.1667, A 0.000, B 0.000, C 0.000 }
gfCNCPoint1[18397] = {X 17.8488, Y 21.8635, Z -2.1667, A 0.000, B 0.000, C 0.000 }
gfCNCPoint1[18398] = {X 17.9274, Y 21.4213, Z -2.1667, A 0.000, B 0.000, C 0.000 }
gfCNCPoint1[18399] = {X 17.8680, Y 20.9760, Z -2.1667, A 0.000, B 0.000, C 0.000 }
gfCNCPoint1[18400] = {X 17.6761, Y 20.5699, Z -2.1667, A 0.000, B 0.000, C 0.000 }
gfCNCPoint1[18401] = {X 17.3699, Y 20.2412, Z -2.1667, A 0.000, B 0.000, C 0.000 }
gfCNCPoint1[18402] = {X 16.4076, Y 19.6747, Z -2.1667, A 0.000, B 0.000, C 0.000 }
gfCNCPoint1[18403] = {X 15.3527, Y 19.3081, Z -2.1667, A 0.000, B 0.000, C 0.000 }
gfCNCPoint1[18404] = {X 13.9979, Y 19.0869, Z -2.1667, A 0.000, B 0.000, C 0.000 }
gfCNCPoint1[18405] = {X 12.6262, Y 19.0320, Z -2.1667, A 0.000, B 0.000, C 0.000 }
gfCNCPoint1[18406] = {X 11.2580, Y 19.1441, Z -2.1667, A 0.000, B 0.000, C 0.000 }
gfCNCPoint1[18407] = {X 10.5678, Y 19.2526, Z -2.1667, A 0.000, B 0.000, C 0.000 }
gfCNCPoint1[18408] = {X 9.5944, Y 19.4791, Z -2.1667, A 0.000, B 0.000, C 0.000 }
gfCNCPoint1[18409] = {X 8.6527, Y 19.8140, Z -2.1667, A 0.000, B 0.000, C 0.000 }
gfCNCPoint1[18410] = {X 7.7548, Y 20.2530, Z -2.1667, A 0.000, B 0.000, C 0.000 }
gfCNCPoint1[18411] = {X 7.7493, Y 20.3318, Z -2.1667, A 0.000, B 0.000, C 0.000 }
gfCNCPoint1[18412] = {X 7.5474, Y 21.2639, Z -2.1667, A 0.000, B 0.000, C 0.000 }
gfCNCPoint1[18413] = {X 7.1385, Y 22.1256, Z -2.1667, A 0.000, B 0.000, C 0.000 }
gfCNCPoint1[18414] = {X 6.5442, Y 22.8714, Z -2.1667, A 0.000, B 0.000, C 0.000 }
gfCNCPoint1[18415] = {X 8.5347, Y 22.6321, Z -2.1667, A 0.000, B 0.000, C 0.000 }
gfCNCPoint1[18416] = {X 10.5350, Y 22.4960, Z -2.1667, A 0.000, B 0.000, C 0.000 }
gfCNCPoint1[18417] = {X 11.1686, Y 22.4709, Z -2.1667, A 0.000, B 0.000, C 0.000 }
gfCNCPoint1[18418] = {X 11.8021, Y 22.4431, Z -2.1667, A 0.000, B 0.000, C 0.000 }
gfCNCPoint1[18419] = {X 15.7666, Y 21.9115, Z -2.1667, A 0.000, B 0.000, C 0.000 }
gfCNCPoint1[18420] = {X 7.8092, Y 22.3582, Z -2.1667, A 0.000, B 0.000, C 0.000 }
gfCNCPoint1[18421] = {X 11.8058, Y 22.5230, Z -2.1667, A 0.000, B 0.000, C 0.000 }
gfCNCPoint1[18422] = {X 14.1394, Y 22.3968, Z -2.1667, A 0.000, B 0.000, C 0.000 }
gfCNCPoint1[18423] = {X 16.4708, Y 22.2334, Z -2.1667, A 0.000, B 0.000, C 0.000 }
gfCNCPoint1[18424] = {X 17.2012, Y 22.1275, Z -2.1667, A 0.000, B 0.000, C 0.000 }
gfCNCPoint1[18425] = {X 17.9113, Y 21.9263, Z -2.1667, A 0.000, B 0.000, C 0.000 }
gfCNCPoint1[18426] = {X 18.0065, Y 21.4520, Z -2.1667, A 0.000, B 0.000, C 0.000 }
gfCNCPoint1[18427] = {X 17.9499, Y 20.9715, Z -2.1667, A 0.000, B 0.000, C 0.000 }
gfCNCPoint1[18428] = {X 17.7472, Y 20.5322, Z -2.1667, A 0.000, B 0.000, C 0.000 }
gfCNCPoint1[18429] = {X 17.4182, Y 20.1774, Z -2.1667, A 0.000, B 0.000, C 0.000 }
gfCNCPoint1[18430] = {X 16.4415, Y 19.6023, Z -2.1667, A 0.000, B 0.000, C 0.000 }
gfCNCPoint1[18431] = {X 15.3709, Y 19.2301, Z -2.1667, A 0.000, B 0.000, C 0.000 }
gfCNCPoint1[18432] = {X 14.0061, Y 19.0073, Z -2.1667, A 0.000, B 0.000, C 0.000 }
gfCNCPoint1[18433] = {X 12.6243, Y 18.9520, Z -2.1667, A 0.000, B 0.000, C 0.000 }
gfCNCPoint1[18434] = {X 11.2461, Y 19.0650, Z -2.1667, A 0.000, B 0.000, C 0.000 }
gfCNCPoint1[18435] = {X 10.5548, Y 19.1737, Z -2.1667, A 0.000, B 0.000, C 0.000 }
gfCNCPoint1[18436] = {X 9.5584, Y 19.4063, Z -2.1667, A 0.000, B 0.000, C 0.000 }
gfCNCPoint1[18437] = {X 8.5953, Y 19.7514, Z -2.1667, A 0.000, B 0.000, C 0.000 }
gfCNCPoint1[18438] = {X 7.6781, Y 20.2045, Z -2.1667, A 0.000, B 0.000, C 0.000 }
gfCNCPoint1[18439] = {X 7.6696, Y 20.3251, Z -2.1667, A 0.000, B 0.000, C 0.000 }
gfCNCPoint1[18440] = {X 7.5230, Y 21.0763, Z -2.1667, A 0.000, B 0.000, C 0.000 }
gfCNCPoint1[18441] = {X 7.2388, Y 21.7869, Z -2.1667, A 0.000, B 0.000, C 0.000 }
gfCNCPoint1[18442] = {X 6.8269, Y 22.4319, Z -2.1667, A 0.000, B 0.000, C 0.000 }
gfCNCPoint1[18443] = {X 6.3017, Y 22.9887, Z -2.1667, A 0.000, B 0.000, C 0.000 }
gfCNCPoint1[18444] = {X 8.4143, Y 22.7240, Z -2.1667, A 0.000, B 0.000, C 0.000 }
gfCNCPoint1[18445] = {X 10.5383, Y 22.5759, Z -2.1667, A 0.000, B 0.000, C 0.000 }
gfCNCPoint1[18446] = {X 11.1721, Y 22.5509, Z -2.1667, A 0.000, B 0.000, C 0.000 }
gfCNCPoint1[18447] = {X 11.8058, Y 22.5230, Z -2.1667, A 0.000, B 0.000, C 0.000 }
gfCNCPoint1[18448] = {X 15.7703, Y 21.9914, Z -2.1667, A 0.000, B 0.000, C 0.000 }
gfCNCPoint1[18449] = {X 11.7345, Y 22.6064, Z -2.1667, A 0.000, B 0.000, C 0.000 }
gfCNCPoint1[18450] = {X 11.8095, Y 22.6030, Z -2.1667, A 0.000, B 0.000, C 0.000 }
gfCNCPoint1[18451] = {X 14.1444, Y 22.4767, Z -2.1667, A 0.000, B 0.000, C 0.000 }
gfCNCPoint1[18452] = {X 16.4770, Y 22.3132, Z -2.1667, A 0.000, B 0.000, C 0.000 }
gfCNCPoint1[18453] = {X 17.2359, Y 22.2019, Z -2.1667, A 0.000, B 0.000, C 0.000 }
gfCNCPoint1[18454] = {X 17.9728, Y 21.9892, Z -2.1667, A 0.000, B 0.000, C 0.000 }
gfCNCPoint1[18455] = {X 18.0851, Y 21.4830, Z -2.1667, A 0.000, B 0.000, C 0.000 }
gfCNCPoint1[18456] = {X 18.0317, Y 20.9672, Z -2.1667, A 0.000, B 0.000, C 0.000 }
gfCNCPoint1[18457] = {X 17.8183, Y 20.4946, Z -2.1667, A 0.000, B 0.000, C 0.000 }
gfCNCPoint1[18458] = {X 17.4665, Y 20.1136, Z -2.1667, A 0.000, B 0.000, C 0.000 }
gfCNCPoint1[18459] = {X 16.4755, Y 19.5298, Z -2.1667, A 0.000, B 0.000, C 0.000 }
gfCNCPoint1[18460] = {X 15.3891, Y 19.1522, Z -2.1667, A 0.000, B 0.000, C 0.000 }
gfCNCPoint1[18461] = {X 14.0143, Y 18.9277, Z -2.1667, A 0.000, B 0.000, C 0.000 }
gfCNCPoint1[18462] = {X 12.6225, Y 18.8720, Z -2.1667, A 0.000, B 0.000, C 0.000 }
gfCNCPoint1[18463] = {X 11.2342, Y 18.9859, Z -2.1667, A 0.000, B 0.000, C 0.000 }
gfCNCPoint1[18464] = {X 10.5417, Y 19.0948, Z -2.1667, A 0.000, B 0.000, C 0.000 }
gfCNCPoint1[18465] = {X 9.5225, Y 19.3335, Z -2.1667, A 0.000, B 0.000, C 0.000 }
gfCNCPoint1[18466] = {X 8.5379, Y 19.6889, Z -2.1667, A 0.000, B 0.000, C 0.000 }
gfCNCPoint1[18467] = {X 7.6013, Y 20.1562, Z -2.1667, A 0.000, B 0.000, C 0.000 }
gfCNCPoint1[18468] = {X 7.5898, Y 20.3183, Z -2.1667, A 0.000, B 0.000, C 0.000 }
gfCNCPoint1[18469] = {X 7.4461, Y 21.0545, Z -2.1667, A 0.000, B 0.000, C 0.000 }
gfCNCPoint1[18470] = {X 7.1674, Y 21.7508, Z -2.1667, A 0.000, B 0.000, C 0.000 }
gfCNCPoint1[18471] = {X 6.7636, Y 22.3830, Z -2.1667, A 0.000, B 0.000, C 0.000 }
gfCNCPoint1[18472] = {X 6.2489, Y 22.9286, Z -2.1667, A 0.000, B 0.000, C 0.000 }
gfCNCPoint1[18473] = {X 6.2076, Y 22.9644, Z -2.1667, A 0.000, B 0.000, C 0.000 }
gfCNCPoint1[18474] = {X 6.1658, Y 22.9996, Z -2.1667, A 0.000, B 0.000, C 0.000 }
gfCNCPoint1[18475] = {X 6.1505, Y 23.0932, Z -2.1667, A 0.000, B 0.000, C 0.000 }
gfCNCPoint1[18476] = {X 6.2322, Y 23.0804, Z -2.1667, A 0.000, B 0.000, C 0.000 }
gfCNCPoint1[18477] = {X 6.3138, Y 23.0678, Z -2.1667, A 0.000, B 0.000, C 0.000 }
gfCNCPoint1[18478] = {X 8.4221, Y 22.8036, Z -2.1667, A 0.000, B 0.000, C 0.000 }
gfCNCPoint1[18479] = {X 10.5417, Y 22.6559, Z -2.1667, A 0.000, B 0.000, C 0.000 }
gfCNCPoint1[18480] = {X 11.1756, Y 22.6308, Z -2.1667, A 0.000, B 0.000, C 0.000 }
gfCNCPoint1[18481] = {X 11.8095, Y 22.6030, Z -2.1667, A 0.000, B 0.000, C 0.000 }
gfCNCPoint1[18482] = {X 11.7174, Y 20.6051, Z -2.1667, A 0.000, B 0.000, C 0.000 }
gfCNCPoint1[18483] = {X 11.7174, Y 20.6051, Z 0.8333, A 0.000, B 0.000, C 0.000 }
gfCNCPoint1[18484] = {X 11.7174, Y 20.6051, Z 11.0000, A 0.000, B 0.000, C 0.000 }
gfCNCPoint1[18485] = {X 11.7112, Y 37.8799, Z 11.0000, A 0.000, B 0.000, C 0.000 }
gfCNCPoint1[18486] = {X 11.7112, Y 37.8799, Z 1.6667, A 0.000, B 0.000, C 0.000 }
gfCNCPoint1[18487] = {X 12.4974, Y 37.9517, Z 1.4551, A 0.000, B 0.000, C 0.000 }
gfCNCPoint1[18488] = {X 14.1383, Y 37.8408, Z 1.0145, A 0.000, B 0.000, C 0.000 }
gfCNCPoint1[18489] = {X 15.7410, Y 37.4723, Z 0.5738, A 0.000, B 0.000, C 0.000 }
gfCNCPoint1[18490] = {X 16.4732, Y 37.1788, Z 0.3624, A 0.000, B 0.000, C 0.000 }
gfCNCPoint1[18491] = {X 17.3049, Y 36.8453, Z 0.1223, A 0.000, B 0.000, C 0.000 }
gfCNCPoint1[18492] = {X 18.2943, Y 36.3175, Z -0.1781, A 0.000, B 0.000, C 0.000 }
gfCNCPoint1[18493] = {X 19.0345, Y 35.8124, Z -0.4183, A 0.000, B 0.000, C 0.000 }
gfCNCPoint1[18494] = {X 19.0577, Y 35.2982, Z -0.5562, A 0.000, B 0.000, C 0.000 }
gfCNCPoint1[18495] = {X 19.2192, Y 34.6347, Z -0.7391, A 0.000, B 0.000, C 0.000 }
gfCNCPoint1[18496] = {X 19.4348, Y 34.1674, Z -0.8770, A 0.000, B 0.000, C 0.000 }
gfCNCPoint1[18497] = {X 18.1966, Y 34.4159, Z -1.2155, A 0.000, B 0.000, C 0.000 }
gfCNCPoint1[18498] = {X 17.3704, Y 34.5281, Z -1.4389, A 0.000, B 0.000, C 0.000 }
gfCNCPoint1[18499] = {X 16.1107, Y 34.6186, Z -1.7773, A 0.000, B 0.000, C 0.000 }
gfCNCPoint1[18500] = {X 15.3861, Y 34.6723, Z -1.9720, A 0.000, B 0.000, C 0.000 }
gfCNCPoint1[18501] = {X 14.6611, Y 34.7219, Z -2.1667, A 0.000, B 0.000, C 0.000 }
gfCNCPoint1[18502] = {X 12.2609, Y 34.8745, Z -2.1667, A 0.000, B 0.000, C 0.000 }
gfCNCPoint1[18503] = {X 9.8594, Y 35.0042, Z -2.1667, A 0.000, B 0.000, C 0.000 }
gfCNCPoint1[18504] = {X 8.7533, Y 35.0947, Z -2.1667, A 0.000, B 0.000, C 0.000 }
gfCNCPoint1[18505] = {X 7.6643, Y 35.3088, Z -2.1667, A 0.000, B 0.000, C 0.000 }
gfCNCPoint1[18506] = {X 7.6546, Y 35.3708, Z -2.1667, A 0.000, B 0.000, C 0.000 }
gfCNCPoint1[18507] = {X 7.6512, Y 35.4334, Z -2.1667, A 0.000, B 0.000, C 0.000 }
gfCNCPoint1[18508] = {X 7.7520, Y 36.0268, Z -2.1667, A 0.000, B 0.000, C 0.000 }
gfCNCPoint1[18509] = {X 8.0469, Y 36.5514, Z -2.1667, A 0.000, B 0.000, C 0.000 }
gfCNCPoint1[18510] = {X 8.5013, Y 36.9460, Z -2.1667, A 0.000, B 0.000, C 0.000 }
gfCNCPoint1[18511] = {X 9.2733, Y 37.3371, Z -2.1667, A 0.000, B 0.000, C 0.000 }
gfCNCPoint1[18512] = {X 10.0947, Y 37.6097, Z -2.1667, A 0.000, B 0.000, C 0.000 }
gfCNCPoint1[18513] = {X 11.3718, Y 37.8469, Z -2.1667, A 0.000, B 0.000, C 0.000 }
gfCNCPoint1[18514] = {X 12.6686, Y 37.9223, Z -2.1667, A 0.000, B 0.000, C 0.000 }
gfCNCPoint1[18515] = {X 13.9646, Y 37.8347, Z -2.1667, A 0.000, B 0.000, C 0.000 }
gfCNCPoint1[18516] = {X 15.2395, Y 37.5856, Z -2.1667, A 0.000, B 0.000, C 0.000 }
gfCNCPoint1[18517] = {X 16.4732, Y 37.1788, Z -2.1667, A 0.000, B 0.000, C 0.000 }
gfCNCPoint1[18518] = {X 17.7910, Y 36.5653, Z -2.1667, A 0.000, B 0.000, C 0.000 }
gfCNCPoint1[18519] = {X 19.0345, Y 35.8124, Z -2.1667, A 0.000, B 0.000, C 0.000 }
gfCNCPoint1[18520] = {X 19.1548, Y 34.9705, Z -2.1667, A 0.000, B 0.000, C 0.000 }
gfCNCPoint1[18521] = {X 19.4348, Y 34.1674, Z -2.1667, A 0.000, B 0.000, C 0.000 }
gfCNCPoint1[18522] = {X 17.7799, Y 34.4455, Z -2.1667, A 0.000, B 0.000, C 0.000 }
gfCNCPoint1[18523] = {X 16.1107, Y 34.6186, Z -2.1667, A 0.000, B 0.000, C 0.000 }
gfCNCPoint1[18524] = {X 15.3860, Y 34.6713, Z -2.1667, A 0.000, B 0.000, C 0.000 }
gfCNCPoint1[18525] = {X 14.6611, Y 34.7219, Z -2.1667, A 0.000, B 0.000, C 0.000 }
gfCNCPoint1[18526] = {X 18.6549, Y 34.7180, Z -2.1667, A 0.000, B 0.000, C 0.000 }
gfCNCPoint1[18527] = {X 14.6557, Y 34.6421, Z -2.1667, A 0.000, B 0.000, C 0.000 }
gfCNCPoint1[18528] = {X 12.2591, Y 34.7945, Z -2.1667, A 0.000, B 0.000, C 0.000 }
gfCNCPoint1[18529] = {X 9.8611, Y 34.9241, Z -2.1667, A 0.000, B 0.000, C 0.000 }
gfCNCPoint1[18530] = {X 8.7204, Y 35.0185, Z -2.1667, A 0.000, B 0.000, C 0.000 }
gfCNCPoint1[18531] = {X 7.5981, Y 35.2432, Z -2.1667, A 0.000, B 0.000, C 0.000 }
gfCNCPoint1[18532] = {X 7.5781, Y 35.3373, Z -2.1667, A 0.000, B 0.000, C 0.000 }
gfCNCPoint1[18533] = {X 7.5712, Y 35.4331, Z -2.1667, A 0.000, B 0.000, C 0.000 }
gfCNCPoint1[18534] = {X 7.6766, Y 36.0535, Z -2.1667, A 0.000, B 0.000, C 0.000 }
gfCNCPoint1[18535] = {X 7.9848, Y 36.6020, Z -2.1667, A 0.000, B 0.000, C 0.000 }
gfCNCPoint1[18536] = {X 8.4600, Y 37.0145, Z -2.1667, A 0.000, B 0.000, C 0.000 }
gfCNCPoint1[18537] = {X 9.2426, Y 37.4109, Z -2.1667, A 0.000, B 0.000, C 0.000 }
gfCNCPoint1[18538] = {X 10.0752, Y 37.6873, Z -2.1667, A 0.000, B 0.000, C 0.000 }
gfCNCPoint1[18539] = {X 11.3622, Y 37.9263, Z -2.1667, A 0.000, B 0.000, C 0.000 }
gfCNCPoint1[18540] = {X 12.6690, Y 38.0023, Z -2.1667, A 0.000, B 0.000, C 0.000 }
gfCNCPoint1[18541] = {X 13.9750, Y 37.9140, Z -2.1667, A 0.000, B 0.000, C 0.000 }
gfCNCPoint1[18542] = {X 15.2598, Y 37.6630, Z -2.1667, A 0.000, B 0.000, C 0.000 }
gfCNCPoint1[18543] = {X 16.5029, Y 37.2530, Z -2.1667, A 0.000, B 0.000, C 0.000 }
gfCNCPoint1[18544] = {X 17.8464, Y 36.6264, Z -2.1667, A 0.000, B 0.000, C 0.000 }
gfCNCPoint1[18545] = {X 19.1128, Y 35.8557, Z -2.1667, A 0.000, B 0.000, C 0.000 }
gfCNCPoint1[18546] = {X 19.2472, Y 34.9310, Z -2.1667, A 0.000, B 0.000, C 0.000 }
gfCNCPoint1[18547] = {X 19.5773, Y 34.0567, Z -2.1667, A 0.000, B 0.000, C 0.000 }
gfCNCPoint1[18548] = {X 17.8491, Y 34.3553, Z -2.1667, A 0.000, B 0.000, C 0.000 }
gfCNCPoint1[18549] = {X 16.1049, Y 34.5388, Z -2.1667, A 0.000, B 0.000, C 0.000 }
gfCNCPoint1[18550] = {X 15.3803, Y 34.5915, Z -2.1667, A 0.000, B 0.000, C 0.000 }
gfCNCPoint1[18551] = {X 14.6557, Y 34.6421, Z -2.1667, A 0.000, B 0.000, C 0.000 }
gfCNCPoint1[18552] = {X 10.7039, Y 35.2617, Z -2.1667, A 0.000, B 0.000, C 0.000 }
gfCNCPoint1[18553] = {X 18.6495, Y 34.6382, Z -2.1667, A 0.000, B 0.000, C 0.000 }
gfCNCPoint1[18554] = {X 14.6502, Y 34.5623, Z -2.1667, A 0.000, B 0.000, C 0.000 }
gfCNCPoint1[18555] = {X 12.2549, Y 34.7146, Z -2.1667, A 0.000, B 0.000, C 0.000 }
gfCNCPoint1[18556] = {X 9.8582, Y 34.8442, Z -2.1667, A 0.000, B 0.000, C 0.000 }
gfCNCPoint1[18557] = {X 8.6869, Y 34.9425, Z -2.1667, A 0.000, B 0.000, C 0.000 }
gfCNCPoint1[18558] = {X 7.5351, Y 35.1771, Z -2.1667, A 0.000, B 0.000, C 0.000 }
gfCNCPoint1[18559] = {X 7.5025, Y 35.3031, Z -2.1667, A 0.000, B 0.000, C 0.000 }
gfCNCPoint1[18560] = {X 7.4912, Y 35.4328, Z -2.1667, A 0.000, B 0.000, C 0.000 }
gfCNCPoint1[18561] = {X 7.6012, Y 36.0802, Z -2.1667, A 0.000, B 0.000, C 0.000 }
gfCNCPoint1[18562] = {X 7.9228, Y 36.6525, Z -2.1667, A 0.000, B 0.000, C 0.000 }
gfCNCPoint1[18563] = {X 8.4186, Y 37.0830, Z -2.1667, A 0.000, B 0.000, C 0.000 }
gfCNCPoint1[18564] = {X 9.2118, Y 37.4848, Z -2.1667, A 0.000, B 0.000, C 0.000 }
gfCNCPoint1[18565] = {X 10.0556, Y 37.7649, Z -2.1667, A 0.000, B 0.000, C 0.000 }
gfCNCPoint1[18566] = {X 11.3525, Y 38.0057, Z -2.1667, A 0.000, B 0.000, C 0.000 }
gfCNCPoint1[18567] = {X 12.6694, Y 38.0823, Z -2.1667, A 0.000, B 0.000, C 0.000 }
gfCNCPoint1[18568] = {X 13.9854, Y 37.9934, Z -2.1667, A 0.000, B 0.000, C 0.000 }
gfCNCPoint1[18569] = {X 15.2800, Y 37.7404, Z -2.1667, A 0.000, B 0.000, C 0.000 }
gfCNCPoint1[18570] = {X 16.5327, Y 37.3273, Z -2.1667, A 0.000, B 0.000, C 0.000 }
gfCNCPoint1[18571] = {X 17.9020, Y 36.6874, Z -2.1667, A 0.000, B 0.000, C 0.000 }
gfCNCPoint1[18572] = {X 19.1915, Y 35.8987, Z -2.1667, A 0.000, B 0.000, C 0.000 }
gfCNCPoint1[18573] = {X 19.2643, Y 35.2207, Z -2.1667, A 0.000, B 0.000, C 0.000 }
gfCNCPoint1[18574] = {X 19.4448, Y 34.5632, Z -2.1667, A 0.000, B 0.000, C 0.000 }
gfCNCPoint1[18575] = {X 19.7284, Y 33.9432, Z -2.1667, A 0.000, B 0.000, C 0.000 }
gfCNCPoint1[18576] = {X 17.9227, Y 34.2641, Z -2.1667, A 0.000, B 0.000, C 0.000 }
gfCNCPoint1[18577] = {X 16.0991, Y 34.4590, Z -2.1667, A 0.000, B 0.000, C 0.000 }
gfCNCPoint1[18578] = {X 15.3747, Y 34.5117, Z -2.1667, A 0.000, B 0.000, C 0.000 }
gfCNCPoint1[18579] = {X 14.6502, Y 34.5623, Z -2.1667, A 0.000, B 0.000, C 0.000 }
gfCNCPoint1[18580] = {X 10.6985, Y 35.1819, Z -2.1667, A 0.000, B 0.000, C 0.000 }
gfCNCPoint1[18581] = {X 18.6440, Y 34.5584, Z -2.1667, A 0.000, B 0.000, C 0.000 }
gfCNCPoint1[18582] = {X 14.6447, Y 34.4824, Z -2.1667, A 0.000, B 0.000, C 0.000 }
gfCNCPoint1[18583] = {X 12.2506, Y 34.6347, Z -2.1667, A 0.000, B 0.000, C 0.000 }
gfCNCPoint1[18584] = {X 9.8552, Y 34.7642, Z -2.1667, A 0.000, B 0.000, C 0.000 }
gfCNCPoint1[18585] = {X 8.6547, Y 34.8663, Z -2.1667, A 0.000, B 0.000, C 0.000 }
gfCNCPoint1[18586] = {X 7.4748, Y 35.1104, Z -2.1667, A 0.000, B 0.000, C 0.000 }
gfCNCPoint1[18587] = {X 7.4276, Y 35.2684, Z -2.1667, A 0.000, B 0.000, C 0.000 }
gfCNCPoint1[18588] = {X 7.4112, Y 35.4326, Z -2.1667, A 0.000, B 0.000, C 0.000 }
gfCNCPoint1[18589] = {X 7.5257, Y 36.1069, Z -2.1667, A 0.000, B 0.000, C 0.000 }
gfCNCPoint1[18590] = {X 7.8608, Y 36.7031, Z -2.1667, A 0.000, B 0.000, C 0.000 }
gfCNCPoint1[18591] = {X 8.3773, Y 37.1515, Z -2.1667, A 0.000, B 0.000, C 0.000 }
gfCNCPoint1[18592] = {X 9.1810, Y 37.5586, Z -2.1667, A 0.000, B 0.000, C 0.000 }
gfCNCPoint1[18593] = {X 10.0361, Y 37.8425, Z -2.1667, A 0.000, B 0.000, C 0.000 }
gfCNCPoint1[18594] = {X 11.3429, Y 38.0851, Z -2.1667, A 0.000, B 0.000, C 0.000 }
gfCNCPoint1[18595] = {X 12.6697, Y 38.1623, Z -2.1667, A 0.000, B 0.000, C 0.000 }
gfCNCPoint1[18596] = {X 13.9958, Y 38.0727, Z -2.1667, A 0.000, B 0.000, C 0.000 }
gfCNCPoint1[18597] = {X 15.3002, Y 37.8178, Z -2.1667, A 0.000, B 0.000, C 0.000 }
gfCNCPoint1[18598] = {X 16.5625, Y 37.4016, Z -2.1667, A 0.000, B 0.000, C 0.000 }
gfCNCPoint1[18599] = {X 17.9579, Y 36.7481, Z -2.1667, A 0.000, B 0.000, C 0.000 }
gfCNCPoint1[18600] = {X 19.2706, Y 35.9412, Z -2.1667, A 0.000, B 0.000, C 0.000 }
gfCNCPoint1[18601] = {X 19.3492, Y 35.2029, Z -2.1667, A 0.000, B 0.000, C 0.000 }
gfCNCPoint1[18602] = {X 19.5579, Y 34.4903, Z -2.1667, A 0.000, B 0.000, C 0.000 }
gfCNCPoint1[18603] = {X 19.8899, Y 33.8262, Z -2.1667, A 0.000, B 0.000, C 0.000 }
gfCNCPoint1[18604] = {X 18.0016, Y 34.1719, Z -2.1667, A 0.000, B 0.000, C 0.000 }
gfCNCPoint1[18605] = {X 16.0932, Y 34.3792, Z -2.1667, A 0.000, B 0.000, C 0.000 }
gfCNCPoint1[18606] = {X 15.3691, Y 34.4319, Z -2.1667, A 0.000, B 0.000, C 0.000 }
gfCNCPoint1[18607] = {X 14.6447, Y 34.4824, Z -2.1667, A 0.000, B 0.000, C 0.000 }
gfCNCPoint1[18608] = {X 10.6930, Y 35.1021, Z -2.1667, A 0.000, B 0.000, C 0.000 }
gfCNCPoint1[18609] = {X 18.6386, Y 34.4786, Z -2.1667, A 0.000, B 0.000, C 0.000 }
gfCNCPoint1[18610] = {X 14.6393, Y 34.4026, Z -2.1667, A 0.000, B 0.000, C 0.000 }
gfCNCPoint1[18611] = {X 12.2464, Y 34.5548, Z -2.1667, A 0.000, B 0.000, C 0.000 }
gfCNCPoint1[18612] = {X 9.8522, Y 34.6843, Z -2.1667, A 0.000, B 0.000, C 0.000 }
gfCNCPoint1[18613] = {X 8.6235, Y 34.7900, Z -2.1667, A 0.000, B 0.000, C 0.000 }
gfCNCPoint1[18614] = {X 7.4166, Y 35.0433, Z -2.1667, A 0.000, B 0.000, C 0.000 }
gfCNCPoint1[18615] = {X 7.3532, Y 35.2332, Z -2.1667, A 0.000, B 0.000, C 0.000 }
gfCNCPoint1[18616] = {X 7.3312, Y 35.4323, Z -2.1667, A 0.000, B 0.000, C 0.000 }
gfCNCPoint1[18617] = {X 7.3980, Y 35.9627, Z -2.1667, A 0.000, B 0.000, C 0.000 }
gfCNCPoint1[18618] = {X 7.5979, Y 36.4586, Z -2.1667, A 0.000, B 0.000, C 0.000 }
gfCNCPoint1[18619] = {X 7.9176, Y 36.8871, Z -2.1667, A 0.000, B 0.000, C 0.000 }
gfCNCPoint1[18620] = {X 8.3360, Y 37.2200, Z -2.1667, A 0.000, B 0.000, C 0.000 }
gfCNCPoint1[18621] = {X 9.1503, Y 37.6325, Z -2.1667, A 0.000, B 0.000, C 0.000 }
gfCNCPoint1[18622] = {X 10.0166, Y 37.9201, Z -2.1667, A 0.000, B 0.000, C 0.000 }
gfCNCPoint1[18623] = {X 11.3332, Y 38.1646, Z -2.1667, A 0.000, B 0.000, C 0.000 }
gfCNCPoint1[18624] = {X 12.6701, Y 38.2423, Z -2.1667, A 0.000, B 0.000, C 0.000 }
gfCNCPoint1[18625] = {X 14.0062, Y 38.1520, Z -2.1667, A 0.000, B 0.000, C 0.000 }
gfCNCPoint1[18626] = {X 15.3205, Y 37.8952, Z -2.1667, A 0.000, B 0.000, C 0.000 }
gfCNCPoint1[18627] = {X 16.5922, Y 37.4758, Z -2.1667, A 0.000, B 0.000, C 0.000 }
gfCNCPoint1[18628] = {X 18.0140, Y 36.8087, Z -2.1667, A 0.000, B 0.000, C 0.000 }
gfCNCPoint1[18629] = {X 19.3501, Y 35.9832, Z -2.1667, A 0.000, B 0.000, C 0.000 }
gfCNCPoint1[18630] = {X 19.4352, Y 35.1814, Z -2.1667, A 0.000, B 0.000, C 0.000 }
gfCNCPoint1[18631] = {X 19.6764, Y 34.4120, Z -2.1667, A 0.000, B 0.000, C 0.000 }
gfCNCPoint1[18632] = {X 20.0642, Y 33.7050, Z -2.1667, A 0.000, B 0.000, C 0.000 }
gfCNCPoint1[18633] = {X 18.0872, Y 34.0785, Z -2.1667, A 0.000, B 0.000, C 0.000 }
gfCNCPoint1[18634] = {X 16.0874, Y 34.2994, Z -2.1667, A 0.000, B 0.000, C 0.000 }
gfCNCPoint1[18635] = {X 15.3634, Y 34.3521, Z -2.1667, A 0.000, B 0.000, C 0.000 }
gfCNCPoint1[18636] = {X 14.6393, Y 34.4026, Z -2.1667, A 0.000, B 0.000, C 0.000 }
gfCNCPoint1[18637] = {X 10.6876, Y 35.0223, Z -2.1667, A 0.000, B 0.000, C 0.000 }
gfCNCPoint1[18638] = {X 14.7703, Y 36.3182, Z -2.1667, A 0.000, B 0.000, C 0.000 }
gfCNCPoint1[18639] = {X 14.6338, Y 34.3228, Z -2.1667, A 0.000, B 0.000, C 0.000 }
gfCNCPoint1[18640] = {X 12.2422, Y 34.4749, Z -2.1667, A 0.000, B 0.000, C 0.000 }
gfCNCPoint1[18641] = {X 9.8492, Y 34.6043, Z -2.1667, A 0.000, B 0.000, C 0.000 }
gfCNCPoint1[18642] = {X 8.5933, Y 34.7136, Z -2.1667, A 0.000, B 0.000, C 0.000 }
gfCNCPoint1[18643] = {X 7.3603, Y 34.9759, Z -2.1667, A 0.000, B 0.000, C 0.000 }
gfCNCPoint1[18644] = {X 7.2793, Y 35.1976, Z -2.1667, A 0.000, B 0.000, C 0.000 }
gfCNCPoint1[18645] = {X 7.2512, Y 35.4320, Z -2.1667, A 0.000, B 0.000, C 0.000 }
gfCNCPoint1[18646] = {X 7.3206, Y 35.9828, Z -2.1667, A 0.000, B 0.000, C 0.000 }
gfCNCPoint1[18647] = {X 7.5281, Y 36.4978, Z -2.1667, A 0.000, B 0.000, C 0.000 }
gfCNCPoint1[18648] = {X 7.8601, Y 36.9428, Z -2.1667, A 0.000, B 0.000, C 0.000 }
gfCNCPoint1[18649] = {X 8.2946, Y 37.2885, Z -2.1667, A 0.000, B 0.000, C 0.000 }
gfCNCPoint1[18650] = {X 9.1195, Y 37.7063, Z -2.1667, A 0.000, B 0.000, C 0.000 }
gfCNCPoint1[18651] = {X 9.9971, Y 37.9977, Z -2.1667, A 0.000, B 0.000, C 0.000 }
gfCNCPoint1[18652] = {X 11.3236, Y 38.2440, Z -2.1667, A 0.000, B 0.000, C 0.000 }
gfCNCPoint1[18653] = {X 12.6705, Y 38.3223, Z -2.1667, A 0.000, B 0.000, C 0.000 }
gfCNCPoint1[18654] = {X 14.0166, Y 38.2313, Z -2.1667, A 0.000, B 0.000, C 0.000 }
gfCNCPoint1[18655] = {X 15.3407, Y 37.9726, Z -2.1667, A 0.000, B 0.000, C 0.000 }
gfCNCPoint1[18656] = {X 16.6220, Y 37.5501, Z -2.1667, A 0.000, B 0.000, C 0.000 }
gfCNCPoint1[18657] = {X 18.0704, Y 36.8692, Z -2.1667, A 0.000, B 0.000, C 0.000 }
gfCNCPoint1[18658] = {X 19.4300, Y 36.0248, Z -2.1667, A 0.000, B 0.000, C 0.000 }
gfCNCPoint1[18659] = {X 19.5226, Y 35.1553, Z -2.1667, A 0.000, B 0.000, C 0.000 }
gfCNCPoint1[18660] = {X 19.8019, Y 34.3266, Z -2.1667, A 0.000, B 0.000, C 0.000 }
gfCNCPoint1[18661] = {X 20.2547, Y 33.5784, Z -2.1667, A 0.000, B 0.000, C 0.000 }
gfCNCPoint1[18662] = {X 18.1811, Y 33.9833, Z -2.1667, A 0.000, B 0.000, C 0.000 }
gfCNCPoint1[18663] = {X 16.0816, Y 34.2196, Z -2.1667, A 0.000, B 0.000, C 0.000 }
gfCNCPoint1[18664] = {X 15.3578, Y 34.2723, Z -2.1667, A 0.000, B 0.000, C 0.000 }
gfCNCPoint1[18665] = {X 14.6338, Y 34.3228, Z -2.1667, A 0.000, B 0.000, C 0.000 }
gfCNCPoint1[18666] = {X 14.7703, Y 36.3182, Z -2.1667, A 0.000, B 0.000, C 0.000 }
gfCNCPoint1[18667] = {X 14.7703, Y 36.3182, Z 0.8333, A 0.000, B 0.000, C 0.000 }
gfCNCPoint1[18668] = {X 14.7703, Y 36.3182, Z 11.0000, A 0.000, B 0.000, C 0.000 }
gfCNCPoint1[18669] = {X 165.6772, Y 73.8165, Z 11.0000, A 0.000, B 0.000, C 0.000 }
gfCNCPoint1[18670] = {X 165.6772, Y 73.8165, Z 1.6667, A 0.000, B 0.000, C 0.000 }
gfCNCPoint1[18671] = {X 161.3996, Y 78.5670, Z -0.0462, A 0.000, B 0.000, C 0.000 }
gfCNCPoint1[18672] = {X 169.3132, Y 78.5670, Z -2.1667, A 0.000, B 0.000, C 0.000 }
gfCNCPoint1[18673] = {X 169.3132, Y 76.1670, Z -2.1667, A 0.000, B 0.000, C 0.000 }
gfCNCPoint1[18674] = {X 171.8361, Y 76.1670, Z -2.1667, A 0.000, B 0.000, C 0.000 }
gfCNCPoint1[18675] = {X 169.3147, Y 73.3634, Z -2.1667, A 0.000, B 0.000, C 0.000 }
gfCNCPoint1[18676] = {X 166.7903, Y 76.1670, Z -2.1667, A 0.000, B 0.000, C 0.000 }
gfCNCPoint1[18677] = {X 169.3132, Y 76.1670, Z -2.1667, A 0.000, B 0.000, C 0.000 }
gfCNCPoint1[18678] = {X 169.3132, Y 78.5670, Z -2.1667, A 0.000, B 0.000, C 0.000 }
gfCNCPoint1[18679] = {X 177.2224, Y 78.5670, Z -2.1667, A 0.000, B 0.000, C 0.000 }
gfCNCPoint1[18680] = {X 169.3158, Y 69.7756, Z -2.1667, A 0.000, B 0.000, C 0.000 }
gfCNCPoint1[18681] = {X 161.3996, Y 78.5670, Z -2.1667, A 0.000, B 0.000, C 0.000 }
gfCNCPoint1[18682] = {X 169.3132, Y 78.5670, Z -2.1667, A 0.000, B 0.000, C 0.000 }
gfCNCPoint1[18683] = {X 169.3132, Y 74.6470, Z -2.1667, A 0.000, B 0.000, C 0.000 }
gfCNCPoint1[18684] = {X 169.3132, Y 78.6470, Z -2.1667, A 0.000, B 0.000, C 0.000 }
gfCNCPoint1[18685] = {X 177.4019, Y 78.6470, Z -2.1667, A 0.000, B 0.000, C 0.000 }
gfCNCPoint1[18686] = {X 169.3159, Y 69.6560, Z -2.1667, A 0.000, B 0.000, C 0.000 }
gfCNCPoint1[18687] = {X 161.2199, Y 78.6470, Z -2.1667, A 0.000, B 0.000, C 0.000 }
gfCNCPoint1[18688] = {X 169.3132, Y 78.6470, Z -2.1667, A 0.000, B 0.000, C 0.000 }
gfCNCPoint1[18689] = {X 169.3132, Y 74.6470, Z -2.1667, A 0.000, B 0.000, C 0.000 }
gfCNCPoint1[18690] = {X 169.3132, Y 74.7270, Z -2.1667, A 0.000, B 0.000, C 0.000 }
gfCNCPoint1[18691] = {X 169.3132, Y 78.7270, Z -2.1667, A 0.000, B 0.000, C 0.000 }
gfCNCPoint1[18692] = {X 177.5814, Y 78.7270, Z -2.1667, A 0.000, B 0.000, C 0.000 }
gfCNCPoint1[18693] = {X 169.3159, Y 69.5364, Z -2.1667, A 0.000, B 0.000, C 0.000 }
gfCNCPoint1[18694] = {X 161.0403, Y 78.7270, Z -2.1667, A 0.000, B 0.000, C 0.000 }
gfCNCPoint1[18695] = {X 169.3132, Y 78.7270, Z -2.1667, A 0.000, B 0.000, C 0.000 }
gfCNCPoint1[18696] = {X 169.3132, Y 74.7270, Z -2.1667, A 0.000, B 0.000, C 0.000 }
gfCNCPoint1[18697] = {X 169.3132, Y 74.8070, Z -2.1667, A 0.000, B 0.000, C 0.000 }
gfCNCPoint1[18698] = {X 169.3132, Y 78.8070, Z -2.1667, A 0.000, B 0.000, C 0.000 }
gfCNCPoint1[18699] = {X 177.7610, Y 78.8070, Z -2.1667, A 0.000, B 0.000, C 0.000 }
gfCNCPoint1[18700] = {X 169.3159, Y 69.4168, Z -2.1667, A 0.000, B 0.000, C 0.000 }
gfCNCPoint1[18701] = {X 160.8606, Y 78.8070, Z -2.1667, A 0.000, B 0.000, C 0.000 }
gfCNCPoint1[18702] = {X 169.3132, Y 78.8070, Z -2.1667, A 0.000, B 0.000, C 0.000 }
gfCNCPoint1[18703] = {X 169.3132, Y 74.8070, Z -2.1667, A 0.000, B 0.000, C 0.000 }
gfCNCPoint1[18704] = {X 169.3132, Y 74.8870, Z -2.1667, A 0.000, B 0.000, C 0.000 }
gfCNCPoint1[18705] = {X 169.3132, Y 78.8870, Z -2.1667, A 0.000, B 0.000, C 0.000 }
gfCNCPoint1[18706] = {X 177.9405, Y 78.8870, Z -2.1667, A 0.000, B 0.000, C 0.000 }
gfCNCPoint1[18707] = {X 169.3160, Y 69.2972, Z -2.1667, A 0.000, B 0.000, C 0.000 }
gfCNCPoint1[18708] = {X 160.6809, Y 78.8870, Z -2.1667, A 0.000, B 0.000, C 0.000 }
gfCNCPoint1[18709] = {X 169.3132, Y 78.8870, Z -2.1667, A 0.000, B 0.000, C 0.000 }
gfCNCPoint1[18710] = {X 169.3132, Y 74.8870, Z -2.1667, A 0.000, B 0.000, C 0.000 }
gfCNCPoint1[18711] = {X 169.3132, Y 74.9670, Z -2.1667, A 0.000, B 0.000, C 0.000 }
gfCNCPoint1[18712] = {X 169.3132, Y 78.9670, Z -2.1667, A 0.000, B 0.000, C 0.000 }
gfCNCPoint1[18713] = {X 178.1201, Y 78.9670, Z -2.1667, A 0.000, B 0.000, C 0.000 }
gfCNCPoint1[18714] = {X 169.3160, Y 69.1776, Z -2.1667, A 0.000, B 0.000, C 0.000 }
gfCNCPoint1[18715] = {X 160.5012, Y 78.9670, Z -2.1667, A 0.000, B 0.000, C 0.000 }
gfCNCPoint1[18716] = {X 169.3132, Y 78.9670, Z -2.1667, A 0.000, B 0.000, C 0.000 }
gfCNCPoint1[18717] = {X 169.3132, Y 74.9670, Z -2.1667, A 0.000, B 0.000, C 0.000 }
gfCNCPoint1[18718] = {X 169.3132, Y 74.9670, Z 0.8333, A 0.000, B 0.000, C 0.000 }
gfCNCPoint1[18719] = {X 169.3132, Y 74.9670, Z 11.0000, A 0.000, B 0.000, C 0.000 }
gfCNCPoint1[18720] = {X 186.2314, Y 37.9128, Z 11.0000, A 0.000, B 0.000, C 0.000 }
gfCNCPoint1[18721] = {X 186.2314, Y 37.9128, Z 1.6667, A 0.000, B 0.000, C 0.000 }
gfCNCPoint1[18722] = {X 187.5937, Y 37.8328, Z 1.3010, A 0.000, B 0.000, C 0.000 }
gfCNCPoint1[18723] = {X 189.4246, Y 37.3844, Z 0.7959, A 0.000, B 0.000, C 0.000 }
gfCNCPoint1[18724] = {X 190.9864, Y 36.7116, Z 0.3403, A 0.000, B 0.000, C 0.000 }
gfCNCPoint1[18725] = {X 191.6931, Y 36.3239, Z 0.1243, A 0.000, B 0.000, C 0.000 }
gfCNCPoint1[18726] = {X 192.4466, Y 35.8120, Z -0.1198, A 0.000, B 0.000, C 0.000 }
gfCNCPoint1[18727] = {X 192.4699, Y 35.2978, Z -0.2577, A 0.000, B 0.000, C 0.000 }
gfCNCPoint1[18728] = {X 192.6317, Y 34.6335, Z -0.4410, A 0.000, B 0.000, C 0.000 }
gfCNCPoint1[18729] = {X 192.8475, Y 34.1662, Z -0.5789, A 0.000, B 0.000, C 0.000 }
gfCNCPoint1[18730] = {X 192.7390, Y 34.1915, Z -0.6087, A 0.000, B 0.000, C 0.000 }
gfCNCPoint1[18731] = {X 191.4110, Y 34.4416, Z -0.9708, A 0.000, B 0.000, C 0.000 }
gfCNCPoint1[18732] = {X 190.5785, Y 34.5487, Z -1.1957, A 0.000, B 0.000, C 0.000 }
gfCNCPoint1[18733] = {X 189.2271, Y 34.6432, Z -1.5587, A 0.000, B 0.000, C 0.000 }
gfCNCPoint1[18734] = {X 186.9625, Y 34.7823, Z -2.1667, A 0.000, B 0.000, C 0.000 }
gfCNCPoint1[18735] = {X 182.5777, Y 35.0515, Z -2.1667, A 0.000, B 0.000, C 0.000 }
gfCNCPoint1[18736] = {X 181.8180, Y 35.1391, Z -2.1667, A 0.000, B 0.000, C 0.000 }
gfCNCPoint1[18737] = {X 181.0720, Y 35.3073, Z -2.1667, A 0.000, B 0.000, C 0.000 }
gfCNCPoint1[18738] = {X 181.0638, Y 35.3818, Z -2.1667, A 0.000, B 0.000, C 0.000 }
gfCNCPoint1[18739] = {X 181.0638, Y 35.4567, Z -2.1667, A 0.000, B 0.000, C 0.000 }
gfCNCPoint1[18740] = {X 181.1565, Y 35.9990, Z -2.1667, A 0.000, B 0.000, C 0.000 }
gfCNCPoint1[18741] = {X 181.4129, Y 36.4858, Z -2.1667, A 0.000, B 0.000, C 0.000 }
gfCNCPoint1[18742] = {X 181.8078, Y 36.8690, Z -2.1667, A 0.000, B 0.000, C 0.000 }
gfCNCPoint1[18743] = {X 182.4210, Y 37.2298, Z -2.1667, A 0.000, B 0.000, C 0.000 }
gfCNCPoint1[18744] = {X 183.0844, Y 37.4873, Z -2.1667, A 0.000, B 0.000, C 0.000 }
gfCNCPoint1[18745] = {X 184.4930, Y 37.8019, Z -2.1667, A 0.000, B 0.000, C 0.000 }
gfCNCPoint1[18746] = {X 185.9317, Y 37.9181, Z -2.1667, A 0.000, B 0.000, C 0.000 }
gfCNCPoint1[18747] = {X 187.3725, Y 37.8334, Z -2.1667, A 0.000, B 0.000, C 0.000 }
gfCNCPoint1[18748] = {X 188.7877, Y 37.5495, Z -2.1667, A 0.000, B 0.000, C 0.000 }
gfCNCPoint1[18749] = {X 190.1497, Y 37.0720, Z -2.1667, A 0.000, B 0.000, C 0.000 }
gfCNCPoint1[18750] = {X 191.3281, Y 36.4966, Z -2.1667, A 0.000, B 0.000, C 0.000 }
gfCNCPoint1[18751] = {X 192.4466, Y 35.8120, Z -2.1667, A 0.000, B 0.000, C 0.000 }
gfCNCPoint1[18752] = {X 192.5671, Y 34.9696, Z -2.1667, A 0.000, B 0.000, C 0.000 }
gfCNCPoint1[18753] = {X 192.8475, Y 34.1662, Z -2.1667, A 0.000, B 0.000, C 0.000 }
gfCNCPoint1[18754] = {X 192.7390, Y 34.1915, Z -2.1667, A 0.000, B 0.000, C 0.000 }
gfCNCPoint1[18755] = {X 190.9896, Y 34.4685, Z -2.1667, A 0.000, B 0.000, C 0.000 }
gfCNCPoint1[18756] = {X 189.2271, Y 34.6432, Z -2.1667, A 0.000, B 0.000, C 0.000 }
gfCNCPoint1[18757] = {X 186.9625, Y 34.7823, Z -2.1667, A 0.000, B 0.000, C 0.000 }
gfCNCPoint1[18758] = {X 190.9562, Y 34.8062, Z -2.1667, A 0.000, B 0.000, C 0.000 }
gfCNCPoint1[18759] = {X 186.9575, Y 34.7024, Z -2.1667, A 0.000, B 0.000, C 0.000 }
gfCNCPoint1[18760] = {X 182.5728, Y 34.9716, Z -2.1667, A 0.000, B 0.000, C 0.000 }
gfCNCPoint1[18761] = {X 181.7804, Y 35.0644, Z -2.1667, A 0.000, B 0.000, C 0.000 }
gfCNCPoint1[18762] = {X 181.0031, Y 35.2438, Z -2.1667, A 0.000, B 0.000, C 0.000 }
gfCNCPoint1[18763] = {X 180.9862, Y 35.3478, Z -2.1667, A 0.000, B 0.000, C 0.000 }
gfCNCPoint1[18764] = {X 180.9837, Y 35.4530, Z -2.1667, A 0.000, B 0.000, C 0.000 }
gfCNCPoint1[18765] = {X 181.0797, Y 36.0219, Z -2.1667, A 0.000, B 0.000, C 0.000 }
gfCNCPoint1[18766] = {X 181.3480, Y 36.5326, Z -2.1667, A 0.000, B 0.000, C 0.000 }
gfCNCPoint1[18767] = {X 181.7618, Y 36.9345, Z -2.1667, A 0.000, B 0.000, C 0.000 }
gfCNCPoint1[18768] = {X 182.3862, Y 37.3018, Z -2.1667, A 0.000, B 0.000, C 0.000 }
gfCNCPoint1[18769] = {X 183.0615, Y 37.5639, Z -2.1667, A 0.000, B 0.000, C 0.000 }
gfCNCPoint1[18770] = {X 184.4810, Y 37.8810, Z -2.1667, A 0.000, B 0.000, C 0.000 }
gfCNCPoint1[18771] = {X 185.9308, Y 37.9981, Z -2.1667, A 0.000, B 0.000, C 0.000 }
gfCNCPoint1[18772] = {X 187.3827, Y 37.9127, Z -2.1667, A 0.000, B 0.000, C 0.000 }
gfCNCPoint1[18773] = {X 188.8088, Y 37.6267, Z -2.1667, A 0.000, B 0.000, C 0.000 }
gfCNCPoint1[18774] = {X 190.1814, Y 37.1455, Z -2.1667, A 0.000, B 0.000, C 0.000 }
gfCNCPoint1[18775] = {X 191.3843, Y 36.5570, Z -2.1667, A 0.000, B 0.000, C 0.000 }
gfCNCPoint1[18776] = {X 192.5249, Y 35.8554, Z -2.1667, A 0.000, B 0.000, C 0.000 }
gfCNCPoint1[18777] = {X 192.6604, Y 34.9269, Z -2.1667, A 0.000, B 0.000, C 0.000 }
gfCNCPoint1[18778] = {X 192.9931, Y 34.0495, Z -2.1667, A 0.000, B 0.000, C 0.000 }
gfCNCPoint1[18779] = {X 192.7316, Y 34.1115, Z -2.1667, A 0.000, B 0.000, C 0.000 }
gfCNCPoint1[18780] = {X 190.9841, Y 34.3885, Z -2.1667, A 0.000, B 0.000, C 0.000 }
gfCNCPoint1[18781] = {X 189.2235, Y 34.5633, Z -2.1667, A 0.000, B 0.000, C 0.000 }
gfCNCPoint1[18782] = {X 186.9575, Y 34.7024, Z -2.1667, A 0.000, B 0.000, C 0.000 }
gfCNCPoint1[18783] = {X 183.0016, Y 35.2946, Z -2.1667, A 0.000, B 0.000, C 0.000 }
gfCNCPoint1[18784] = {X 190.9513, Y 34.7263, Z -2.1667, A 0.000, B 0.000, C 0.000 }
gfCNCPoint1[18785] = {X 186.9526, Y 34.6226, Z -2.1667, A 0.000, B 0.000, C 0.000 }
gfCNCPoint1[18786] = {X 182.5679, Y 34.8918, Z -2.1667, A 0.000, B 0.000, C 0.000 }
gfCNCPoint1[18787] = {X 181.7444, Y 34.9895, Z -2.1667, A 0.000, B 0.000, C 0.000 }
gfCNCPoint1[18788] = {X 180.9373, Y 35.1798, Z -2.1667, A 0.000, B 0.000, C 0.000 }
gfCNCPoint1[18789] = {X 180.9092, Y 35.3161, Z -2.1667, A 0.000, B 0.000, C 0.000 }
gfCNCPoint1[18790] = {X 180.9037, Y 35.4552, Z -2.1667, A 0.000, B 0.000, C 0.000 }
gfCNCPoint1[18791] = {X 181.0042, Y 36.0483, Z -2.1667, A 0.000, B 0.000, C 0.000 }
gfCNCPoint1[18792] = {X 181.2842, Y 36.5808, Z -2.1667, A 0.000, B 0.000, C 0.000 }
gfCNCPoint1[18793] = {X 181.7158, Y 36.9999, Z -2.1667, A 0.000, B 0.000, C 0.000 }
gfCNCPoint1[18794] = {X 182.3513, Y 37.3738, Z -2.1667, A 0.000, B 0.000, C 0.000 }
gfCNCPoint1[18795] = {X 183.0387, Y 37.6406, Z -2.1667, A 0.000, B 0.000, C 0.000 }
gfCNCPoint1[18796] = {X 184.4690, Y 37.9601, Z -2.1667, A 0.000, B 0.000, C 0.000 }
gfCNCPoint1[18797] = {X 185.9299, Y 38.0781, Z -2.1667, A 0.000, B 0.000, C 0.000 }
gfCNCPoint1[18798] = {X 187.3930, Y 37.9921, Z -2.1667, A 0.000, B 0.000, C 0.000 }
gfCNCPoint1[18799] = {X 188.8300, Y 37.7038, Z -2.1667, A 0.000, B 0.000, C 0.000 }
gfCNCPoint1[18800] = {X 190.2130, Y 37.2190, Z -2.1667, A 0.000, B 0.000, C 0.000 }
gfCNCPoint1[18801] = {X 191.4407, Y 36.6173, Z -2.1667, A 0.000, B 0.000, C 0.000 }
gfCNCPoint1[18802] = {X 192.6036, Y 35.8985, Z -2.1667, A 0.000, B 0.000, C 0.000 }
gfCNCPoint1[18803] = {X 192.6774, Y 35.2159, Z -2.1667, A 0.000, B 0.000, C 0.000 }
gfCNCPoint1[18804] = {X 192.8603, Y 34.5542, Z -2.1667, A 0.000, B 0.000, C 0.000 }
gfCNCPoint1[18805] = {X 193.1476, Y 33.9306, Z -2.1667, A 0.000, B 0.000, C 0.000 }
gfCNCPoint1[18806] = {X 192.7149, Y 34.0332, Z -2.1667, A 0.000, B 0.000, C 0.000 }
gfCNCPoint1[18807] = {X 190.9732, Y 34.3093, Z -2.1667, A 0.000, B 0.000, C 0.000 }
gfCNCPoint1[18808] = {X 189.2183, Y 34.4834, Z -2.1667, A 0.000, B 0.000, C 0.000 }
gfCNCPoint1[18809] = {X 186.9526, Y 34.6226, Z -2.1667, A 0.000, B 0.000, C 0.000 }
gfCNCPoint1[18810] = {X 182.9967, Y 35.2147, Z -2.1667, A 0.000, B 0.000, C 0.000 }
gfCNCPoint1[18811] = {X 190.9464, Y 34.6465, Z -2.1667, A 0.000, B 0.000, C 0.000 }
gfCNCPoint1[18812] = {X 186.9477, Y 34.5427, Z -2.1667, A 0.000, B 0.000, C 0.000 }
gfCNCPoint1[18813] = {X 182.5630, Y 34.8119, Z -2.1667, A 0.000, B 0.000, C 0.000 }
gfCNCPoint1[18814] = {X 181.7096, Y 34.9144, Z -2.1667, A 0.000, B 0.000, C 0.000 }
gfCNCPoint1[18815] = {X 180.8740, Y 35.1152, Z -2.1667, A 0.000, B 0.000, C 0.000 }
gfCNCPoint1[18816] = {X 180.8328, Y 35.2839, Z -2.1667, A 0.000, B 0.000, C 0.000 }
gfCNCPoint1[18817] = {X 180.8237, Y 35.4572, Z -2.1667, A 0.000, B 0.000, C 0.000 }
gfCNCPoint1[18818] = {X 180.9287, Y 36.0747, Z -2.1667, A 0.000, B 0.000, C 0.000 }
gfCNCPoint1[18819] = {X 181.2204, Y 36.6291, Z -2.1667, A 0.000, B 0.000, C 0.000 }
gfCNCPoint1[18820] = {X 181.6698, Y 37.0654, Z -2.1667, A 0.000, B 0.000, C 0.000 }
gfCNCPoint1[18821] = {X 182.3164, Y 37.4458, Z -2.1667, A 0.000, B 0.000, C 0.000 }
gfCNCPoint1[18822] = {X 183.0159, Y 37.7173, Z -2.1667, A 0.000, B 0.000, C 0.000 }
gfCNCPoint1[18823] = {X 184.4571, Y 38.0392, Z -2.1667, A 0.000, B 0.000, C 0.000 }
gfCNCPoint1[18824] = {X 185.9290, Y 38.1580, Z -2.1667, A 0.000, B 0.000, C 0.000 }
gfCNCPoint1[18825] = {X 187.4032, Y 38.0714, Z -2.1667, A 0.000, B 0.000, C 0.000 }
gfCNCPoint1[18826] = {X 188.8511, Y 37.7810, Z -2.1667, A 0.000, B 0.000, C 0.000 }
gfCNCPoint1[18827] = {X 190.2447, Y 37.2924, Z -2.1667, A 0.000, B 0.000, C 0.000 }
gfCNCPoint1[18828] = {X 191.4973, Y 36.6774, Z -2.1667, A 0.000, B 0.000, C 0.000 }
gfCNCPoint1[18829] = {X 192.6827, Y 35.9411, Z -2.1667, A 0.000, B 0.000, C 0.000 }
gfCNCPoint1[18830] = {X 192.7627, Y 35.1963, Z -2.1667, A 0.000, B 0.000, C 0.000 }
gfCNCPoint1[18831] = {X 192.9749, Y 34.4780, Z -2.1667, A 0.000, B 0.000, C 0.000 }
gfCNCPoint1[18832] = {X 193.3125, Y 33.8093, Z -2.1667, A 0.000, B 0.000, C 0.000 }
gfCNCPoint1[18833] = {X 192.6983, Y 33.9550, Z -2.1667, A 0.000, B 0.000, C 0.000 }
gfCNCPoint1[18834] = {X 190.9622, Y 34.2301, Z -2.1667, A 0.000, B 0.000, C 0.000 }
gfCNCPoint1[18835] = {X 189.2130, Y 34.4036, Z -2.1667, A 0.000, B 0.000, C 0.000 }
gfCNCPoint1[18836] = {X 186.9477, Y 34.5427, Z -2.1667, A 0.000, B 0.000, C 0.000 }
gfCNCPoint1[18837] = {X 182.9918, Y 35.1349, Z -2.1667, A 0.000, B 0.000, C 0.000 }
gfCNCPoint1[18838] = {X 190.9415, Y 34.5666, Z -2.1667, A 0.000, B 0.000, C 0.000 }
gfCNCPoint1[18839] = {X 186.9428, Y 34.4629, Z -2.1667, A 0.000, B 0.000, C 0.000 }
gfCNCPoint1[18840] = {X 182.5580, Y 34.7321, Z -2.1667, A 0.000, B 0.000, C 0.000 }
gfCNCPoint1[18841] = {X 181.6759, Y 34.8392, Z -2.1667, A 0.000, B 0.000, C 0.000 }
gfCNCPoint1[18842] = {X 180.8127, Y 35.0503, Z -2.1667, A 0.000, B 0.000, C 0.000 }
gfCNCPoint1[18843] = {X 180.7570, Y 35.2512, Z -2.1667, A 0.000, B 0.000, C 0.000 }
gfCNCPoint1[18844] = {X 180.7438, Y 35.4593, Z -2.1667, A 0.000, B 0.000, C 0.000 }
gfCNCPoint1[18845] = {X 180.8532, Y 36.1012, Z -2.1667, A 0.000, B 0.000, C 0.000 }
gfCNCPoint1[18846] = {X 181.1565, Y 36.6773, Z -2.1667, A 0.000, B 0.000, C 0.000 }
gfCNCPoint1[18847] = {X 181.6238, Y 37.1308, Z -2.1667, A 0.000, B 0.000, C 0.000 }
gfCNCPoint1[18848] = {X 182.2816, Y 37.5178, Z -2.1667, A 0.000, B 0.000, C 0.000 }
gfCNCPoint1[18849] = {X 182.9930, Y 37.7940, Z -2.1667, A 0.000, B 0.000, C 0.000 }
gfCNCPoint1[18850] = {X 184.4451, Y 38.1183, Z -2.1667, A 0.000, B 0.000, C 0.000 }
gfCNCPoint1[18851] = {X 185.9282, Y 38.2380, Z -2.1667, A 0.000, B 0.000, C 0.000 }
gfCNCPoint1[18852] = {X 187.4135, Y 38.1508, Z -2.1667, A 0.000, B 0.000, C 0.000 }
gfCNCPoint1[18853] = {X 188.8723, Y 37.8582, Z -2.1667, A 0.000, B 0.000, C 0.000 }
gfCNCPoint1[18854] = {X 190.2764, Y 37.3659, Z -2.1667, A 0.000, B 0.000, C 0.000 }
gfCNCPoint1[18855] = {X 191.5542, Y 36.7373, Z -2.1667, A 0.000, B 0.000, C 0.000 }
gfCNCPoint1[18856] = {X 192.7622, Y 35.9833, Z -2.1667, A 0.000, B 0.000, C 0.000 }
gfCNCPoint1[18857] = {X 192.8359, Y 35.2387, Z -2.1667, A 0.000, B 0.000, C 0.000 }
gfCNCPoint1[18858] = {X 193.0443, Y 34.5201, Z -2.1667, A 0.000, B 0.000, C 0.000 }
gfCNCPoint1[18859] = {X 193.3804, Y 33.8517, Z -2.1667, A 0.000, B 0.000, C 0.000 }
gfCNCPoint1[18860] = {X 193.4232, Y 33.7844, Z -2.1667, A 0.000, B 0.000, C 0.000 }
gfCNCPoint1[18861] = {X 193.4674, Y 33.7180, Z -2.1667, A 0.000, B 0.000, C 0.000 }
gfCNCPoint1[18862] = {X 193.3655, Y 33.7146, Z -2.1667, A 0.000, B 0.000, C 0.000 }
gfCNCPoint1[18863] = {X 192.6816, Y 33.8767, Z -2.1667, A 0.000, B 0.000, C 0.000 }
gfCNCPoint1[18864] = {X 190.9512, Y 34.1508, Z -2.1667, A 0.000, B 0.000, C 0.000 }
gfCNCPoint1[18865] = {X 189.2078, Y 34.3238, Z -2.1667, A 0.000, B 0.000, C 0.000 }
gfCNCPoint1[18866] = {X 186.9428, Y 34.4629, Z -2.1667, A 0.000, B 0.000, C 0.000 }
gfCNCPoint1[18867] = {X 182.9869, Y 35.0550, Z -2.1667, A 0.000, B 0.000, C 0.000 }
gfCNCPoint1[18868] = {X 190.9366, Y 34.4868, Z -2.1667, A 0.000, B 0.000, C 0.000 }
gfCNCPoint1[18869] = {X 186.9379, Y 34.3830, Z -2.1667, A 0.000, B 0.000, C 0.000 }
gfCNCPoint1[18870] = {X 182.5531, Y 34.6522, Z -2.1667, A 0.000, B 0.000, C 0.000 }
gfCNCPoint1[18871] = {X 181.6430, Y 34.7639, Z -2.1667, A 0.000, B 0.000, C 0.000 }
gfCNCPoint1[18872] = {X 180.7531, Y 34.9851, Z -2.1667, A 0.000, B 0.000, C 0.000 }
gfCNCPoint1[18873] = {X 180.6816, Y 35.2182, Z -2.1667, A 0.000, B 0.000, C 0.000 }
gfCNCPoint1[18874] = {X 180.6638, Y 35.4613, Z -2.1667, A 0.000, B 0.000, C 0.000 }
gfCNCPoint1[18875] = {X 180.7777, Y 36.1276, Z -2.1667, A 0.000, B 0.000, C 0.000 }
gfCNCPoint1[18876] = {X 181.0927, Y 36.7256, Z -2.1667, A 0.000, B 0.000, C 0.000 }
gfCNCPoint1[18877] = {X 181.5778, Y 37.1963, Z -2.1667, A 0.000, B 0.000, C 0.000 }
gfCNCPoint1[18878] = {X 182.2467, Y 37.5898, Z -2.1667, A 0.000, B 0.000, C 0.000 }
gfCNCPoint1[18879] = {X 182.9702, Y 37.8706, Z -2.1667, A 0.000, B 0.000, C 0.000 }
gfCNCPoint1[18880] = {X 184.4331, Y 38.1974, Z -2.1667, A 0.000, B 0.000, C 0.000 }
gfCNCPoint1[18881] = {X 185.9273, Y 38.3180, Z -2.1667, A 0.000, B 0.000, C 0.000 }
gfCNCPoint1[18882] = {X 187.4237, Y 38.2301, Z -2.1667, A 0.000, B 0.000, C 0.000 }
gfCNCPoint1[18883] = {X 188.8934, Y 37.9353, Z -2.1667, A 0.000, B 0.000, C 0.000 }
gfCNCPoint1[18884] = {X 190.3080, Y 37.4394, Z -2.1667, A 0.000, B 0.000, C 0.000 }
gfCNCPoint1[18885] = {X 191.6113, Y 36.7970, Z -2.1667, A 0.000, B 0.000, C 0.000 }
gfCNCPoint1[18886] = {X 192.8422, Y 36.0250, Z -2.1667, A 0.000, B 0.000, C 0.000 }
gfCNCPoint1[18887] = {X 192.9290, Y 35.1818, Z -2.1667, A 0.000, B 0.000, C 0.000 }
gfCNCPoint1[18888] = {X 193.1917, Y 34.3757, Z -2.1667, A 0.000, B 0.000, C 0.000 }
gfCNCPoint1[18889] = {X 193.6183, Y 33.6431, Z -2.1667, A 0.000, B 0.000, C 0.000 }
gfCNCPoint1[18890] = {X 193.3575, Y 33.6342, Z -2.1667, A 0.000, B 0.000, C 0.000 }
gfCNCPoint1[18891] = {X 192.6650, Y 33.7984, Z -2.1667, A 0.000, B 0.000, C 0.000 }
gfCNCPoint1[18892] = {X 190.9403, Y 34.0716, Z -2.1667, A 0.000, B 0.000, C 0.000 }
gfCNCPoint1[18893] = {X 189.2026, Y 34.2440, Z -2.1667, A 0.000, B 0.000, C 0.000 }
gfCNCPoint1[18894] = {X 186.9379, Y 34.3830, Z -2.1667, A 0.000, B 0.000, C 0.000 }
gfCNCPoint1[18895] = {X 182.9455, Y 34.6281, Z -2.1667, A 0.000, B 0.000, C 0.000 }
gfCNCPoint1[18896] = {X 182.9455, Y 34.6281, Z 0.8333, A 0.000, B 0.000, C 0.000 }
gfCNCPoint1[18897] = {X 182.9455, Y 34.6281, Z 11.0000, A 0.000, B 0.000, C 0.000 }
gfCNCPoint1[18898] = {X 188.4943, Y 19.4651, Z 11.0000, A 0.000, B 0.000, C 0.000 }
gfCNCPoint1[18899] = {X 188.4943, Y 19.4651, Z 1.6667, A 0.000, B 0.000, C 0.000 }
gfCNCPoint1[18900] = {X 188.3890, Y 19.4279, Z 1.6368, A 0.000, B 0.000, C 0.000 }
gfCNCPoint1[18901] = {X 187.7714, Y 19.3589, Z 1.4702, A 0.000, B 0.000, C 0.000 }
gfCNCPoint1[18902] = {X 186.9109, Y 19.2589, Z 1.2381, A 0.000, B 0.000, C 0.000 }
gfCNCPoint1[18903] = {X 184.5930, Y 19.3664, Z 0.6164, A 0.000, B 0.000, C 0.000 }
gfCNCPoint1[18904] = {X 183.7431, Y 19.5461, Z 0.3836, A 0.000, B 0.000, C 0.000 }
gfCNCPoint1[18905] = {X 183.0411, Y 19.6901, Z 0.1916, A 0.000, B 0.000, C 0.000 }
gfCNCPoint1[18906] = {X 182.0259, Y 20.0596, Z -0.0979, A 0.000, B 0.000, C 0.000 }
gfCNCPoint1[18907] = {X 181.3956, Y 20.4005, Z -0.2899, A 0.000, B 0.000, C 0.000 }
gfCNCPoint1[18908] = {X 181.3397, Y 20.9122, Z -0.4278, A 0.000, B 0.000, C 0.000 }
gfCNCPoint1[18909] = {X 180.8641, Y 22.1276, Z -0.7775, A 0.000, B 0.000, C 0.000 }
gfCNCPoint1[18910] = {X 180.5578, Y 22.5413, Z -0.9155, A 0.000, B 0.000, C 0.000 }
gfCNCPoint1[18911] = {X 182.2905, Y 22.3353, Z -1.3830, A 0.000, B 0.000, C 0.000 }
gfCNCPoint1[18912] = {X 182.5945, Y 22.3106, Z -1.4647, A 0.000, B 0.000, C 0.000 }
gfCNCPoint1[18913] = {X 184.3414, Y 22.2345, Z -1.9332, A 0.000, B 0.000, C 0.000 }
gfCNCPoint1[18914] = {X 184.7767, Y 22.2194, Z -2.0500, A 0.000, B 0.000, C 0.000 }
gfCNCPoint1[18915] = {X 185.2119, Y 22.2011, Z -2.1667, A 0.000, B 0.000, C 0.000 }
gfCNCPoint1[18916] = {X 187.5426, Y 22.0785, Z -2.1667, A 0.000, B 0.000, C 0.000 }
gfCNCPoint1[18917] = {X 189.8704, Y 21.9077, Z -2.1667, A 0.000, B 0.000, C 0.000 }
gfCNCPoint1[18918] = {X 190.4721, Y 21.8319, Z -2.1667, A 0.000, B 0.000, C 0.000 }
gfCNCPoint1[18919] = {X 191.0593, Y 21.6805, Z -2.1667, A 0.000, B 0.000, C 0.000 }
gfCNCPoint1[18920] = {X 191.0691, Y 21.1637, Z -2.1667, A 0.000, B 0.000, C 0.000 }
gfCNCPoint1[18921] = {X 190.8729, Y 20.6855, Z -2.1667, A 0.000, B 0.000, C 0.000 }
gfCNCPoint1[18922] = {X 190.5028, Y 20.3246, Z -2.1667, A 0.000, B 0.000, C 0.000 }
gfCNCPoint1[18923] = {X 189.6452, Y 19.8645, Z -2.1667, A 0.000, B 0.000, C 0.000 }
gfCNCPoint1[18924] = {X 188.7277, Y 19.5401, Z -2.1667, A 0.000, B 0.000, C 0.000 }
gfCNCPoint1[18925] = {X 187.7714, Y 19.3589, Z -2.1667, A 0.000, B 0.000, C 0.000 }
gfCNCPoint1[18926] = {X 186.4245, Y 19.2758, Z -2.1667, A 0.000, B 0.000, C 0.000 }
gfCNCPoint1[18927] = {X 185.0765, Y 19.3384, Z -2.1667, A 0.000, B 0.000, C 0.000 }
gfCNCPoint1[18928] = {X 183.7431, Y 19.5461, Z -2.1667, A 0.000, B 0.000, C 0.000 }
gfCNCPoint1[18929] = {X 182.5379, Y 19.8870, Z -2.1667, A 0.000, B 0.000, C 0.000 }
gfCNCPoint1[18930] = {X 181.3956, Y 20.4005, Z -2.1667, A 0.000, B 0.000, C 0.000 }
gfCNCPoint1[18931] = {X 181.2442, Y 21.1598, Z -2.1667, A 0.000, B 0.000, C 0.000 }
gfCNCPoint1[18932] = {X 180.9620, Y 21.8809, Z -2.1667, A 0.000, B 0.000, C 0.000 }
gfCNCPoint1[18933] = {X 180.5578, Y 22.5413, Z -2.1667, A 0.000, B 0.000, C 0.000 }
gfCNCPoint1[18934] = {X 182.4467, Y 22.3525, Z -2.1667, A 0.000, B 0.000, C 0.000 }
gfCNCPoint1[18935] = {X 184.3414, Y 22.2345, Z -2.1667, A 0.000, B 0.000, C 0.000 }
gfCNCPoint1[18936] = {X 184.7767, Y 22.2186, Z -2.1667, A 0.000, B 0.000, C 0.000 }
gfCNCPoint1[18937] = {X 185.2119, Y 22.2011, Z -2.1667, A 0.000, B 0.000, C 0.000 }
gfCNCPoint1[18938] = {X 181.2193, Y 22.1009, Z -2.1667, A 0.000, B 0.000, C 0.000 }
gfCNCPoint1[18939] = {X 185.2153, Y 22.2810, Z -2.1667, A 0.000, B 0.000, C 0.000 }
gfCNCPoint1[18940] = {X 187.5451, Y 22.1584, Z -2.1667, A 0.000, B 0.000, C 0.000 }
gfCNCPoint1[18941] = {X 189.8719, Y 21.9877, Z -2.1667, A 0.000, B 0.000, C 0.000 }
gfCNCPoint1[18942] = {X 190.5073, Y 21.9065, Z -2.1667, A 0.000, B 0.000, C 0.000 }
gfCNCPoint1[18943] = {X 191.1265, Y 21.7424, Z -2.1667, A 0.000, B 0.000, C 0.000 }
gfCNCPoint1[18944] = {X 191.1530, Y 21.1789, Z -2.1667, A 0.000, B 0.000, C 0.000 }
gfCNCPoint1[18945] = {X 190.9476, Y 20.6534, Z -2.1667, A 0.000, B 0.000, C 0.000 }
gfCNCPoint1[18946] = {X 190.5459, Y 20.2572, Z -2.1667, A 0.000, B 0.000, C 0.000 }
gfCNCPoint1[18947] = {X 189.6781, Y 19.7916, Z -2.1667, A 0.000, B 0.000, C 0.000 }
gfCNCPoint1[18948] = {X 188.7497, Y 19.4631, Z -2.1667, A 0.000, B 0.000, C 0.000 }
gfCNCPoint1[18949] = {X 187.7821, Y 19.2796, Z -2.1667, A 0.000, B 0.000, C 0.000 }
gfCNCPoint1[18950] = {X 186.4269, Y 19.1958, Z -2.1667, A 0.000, B 0.000, C 0.000 }
gfCNCPoint1[18951] = {X 185.0705, Y 19.2586, Z -2.1667, A 0.000, B 0.000, C 0.000 }
gfCNCPoint1[18952] = {X 183.7289, Y 19.4673, Z -2.1667, A 0.000, B 0.000, C 0.000 }
gfCNCPoint1[18953] = {X 182.4923, Y 19.8186, Z -2.1667, A 0.000, B 0.000, C 0.000 }
gfCNCPoint1[18954] = {X 181.3216, Y 20.3497, Z -2.1667, A 0.000, B 0.000, C 0.000 }
gfCNCPoint1[18955] = {X 181.1582, Y 21.1710, Z -2.1667, A 0.000, B 0.000, C 0.000 }
gfCNCPoint1[18956] = {X 180.8394, Y 21.9454, Z -2.1667, A 0.000, B 0.000, C 0.000 }
gfCNCPoint1[18957] = {X 180.3773, Y 22.6437, Z -2.1667, A 0.000, B 0.000, C 0.000 }
gfCNCPoint1[18958] = {X 182.3567, Y 22.4401, Z -2.1667, A 0.000, B 0.000, C 0.000 }
gfCNCPoint1[18959] = {X 184.3427, Y 22.3145, Z -2.1667, A 0.000, B 0.000, C 0.000 }
gfCNCPoint1[18960] = {X 184.7790, Y 22.2986, Z -2.1667, A 0.000, B 0.000, C 0.000 }
gfCNCPoint1[18961] = {X 185.2153, Y 22.2810, Z -2.1667, A 0.000, B 0.000, C 0.000 }
gfCNCPoint1[18962] = {X 189.1818, Y 21.7645, Z -2.1667, A 0.000, B 0.000, C 0.000 }
gfCNCPoint1[18963] = {X 181.2227, Y 22.1808, Z -2.1667, A 0.000, B 0.000, C 0.000 }
gfCNCPoint1[18964] = {X 185.2186, Y 22.3609, Z -2.1667, A 0.000, B 0.000, C 0.000 }
gfCNCPoint1[18965] = {X 187.5497, Y 22.2383, Z -2.1667, A 0.000, B 0.000, C 0.000 }
gfCNCPoint1[18966] = {X 189.8776, Y 22.0675, Z -2.1667, A 0.000, B 0.000, C 0.000 }
gfCNCPoint1[18967] = {X 190.5439, Y 21.9808, Z -2.1667, A 0.000, B 0.000, C 0.000 }
gfCNCPoint1[18968] = {X 191.1923, Y 21.8045, Z -2.1667, A 0.000, B 0.000, C 0.000 }
gfCNCPoint1[18969] = {X 191.2500, Y 21.3479, Z -2.1667, A 0.000, B 0.000, C 0.000 }
gfCNCPoint1[18970] = {X 191.1602, Y 20.8964, Z -2.1667, A 0.000, B 0.000, C 0.000 }
gfCNCPoint1[18971] = {X 190.9320, Y 20.4967, Z -2.1667, A 0.000, B 0.000, C 0.000 }
gfCNCPoint1[18972] = {X 190.5890, Y 20.1898, Z -2.1667, A 0.000, B 0.000, C 0.000 }
gfCNCPoint1[18973] = {X 189.7105, Y 19.7184, Z -2.1667, A 0.000, B 0.000, C 0.000 }
gfCNCPoint1[18974] = {X 188.7705, Y 19.3859, Z -2.1667, A 0.000, B 0.000, C 0.000 }
gfCNCPoint1[18975] = {X 187.7910, Y 19.2001, Z -2.1667, A 0.000, B 0.000, C 0.000 }
gfCNCPoint1[18976] = {X 186.4273, Y 19.1158, Z -2.1667, A 0.000, B 0.000, C 0.000 }
gfCNCPoint1[18977] = {X 185.0624, Y 19.1790, Z -2.1667, A 0.000, B 0.000, C 0.000 }
gfCNCPoint1[18978] = {X 183.7123, Y 19.3891, Z -2.1667, A 0.000, B 0.000, C 0.000 }
gfCNCPoint1[18979] = {X 182.4466, Y 19.7501, Z -2.1667, A 0.000, B 0.000, C 0.000 }
gfCNCPoint1[18980] = {X 181.2497, Y 20.2979, Z -2.1667, A 0.000, B 0.000, C 0.000 }
gfCNCPoint1[18981] = {X 181.2398, Y 20.3520, Z -2.1667, A 0.000, B 0.000, C 0.000 }
gfCNCPoint1[18982] = {X 181.0789, Y 21.1543, Z -2.1667, A 0.000, B 0.000, C 0.000 }
gfCNCPoint1[18983] = {X 180.7668, Y 21.9108, Z -2.1667, A 0.000, B 0.000, C 0.000 }
gfCNCPoint1[18984] = {X 180.3151, Y 22.5933, Z -2.1667, A 0.000, B 0.000, C 0.000 }
gfCNCPoint1[18985] = {X 180.2504, Y 22.6712, Z -2.1667, A 0.000, B 0.000, C 0.000 }
gfCNCPoint1[18986] = {X 180.1838, Y 22.7476, Z -2.1667, A 0.000, B 0.000, C 0.000 }
gfCNCPoint1[18987] = {X 180.1889, Y 22.7478, Z -2.1667, A 0.000, B 0.000, C 0.000 }
gfCNCPoint1[18988] = {X 180.2880, Y 22.7353, Z -2.1667, A 0.000, B 0.000, C 0.000 }
gfCNCPoint1[18989] = {X 180.3870, Y 22.7231, Z -2.1667, A 0.000, B 0.000, C 0.000 }
gfCNCPoint1[18990] = {X 182.3632, Y 22.5199, Z -2.1667, A 0.000, B 0.000, C 0.000 }
gfCNCPoint1[18991] = {X 184.3458, Y 22.3944, Z -2.1667, A 0.000, B 0.000, C 0.000 }
gfCNCPoint1[18992] = {X 184.7823, Y 22.3785, Z -2.1667, A 0.000, B 0.000, C 0.000 }
gfCNCPoint1[18993] = {X 185.2186, Y 22.3609, Z -2.1667, A 0.000, B 0.000, C 0.000 }
gfCNCPoint1[18994] = {X 189.1852, Y 21.8444, Z -2.1667, A 0.000, B 0.000, C 0.000 }
gfCNCPoint1[18995] = {X 181.2261, Y 22.2608, Z -2.1667, A 0.000, B 0.000, C 0.000 }
gfCNCPoint1[18996] = {X 185.2220, Y 22.4408, Z -2.1667, A 0.000, B 0.000, C 0.000 }
gfCNCPoint1[18997] = {X 187.5542, Y 22.3182, Z -2.1667, A 0.000, B 0.000, C 0.000 }
gfCNCPoint1[18998] = {X 189.8834, Y 22.1473, Z -2.1667, A 0.000, B 0.000, C 0.000 }
gfCNCPoint1[18999] = {X 190.5799, Y 22.0552, Z -2.1667, A 0.000, B 0.000, C 0.000 }
gfCNCPoint1[19000] = {X 191.2567, Y 21.8667, Z -2.1667, A 0.000, B 0.000, C 0.000 }
gfCNCPoint1[19001] = {X 191.3308, Y 21.3761, Z -2.1667, A 0.000, B 0.000, C 0.000 }
gfCNCPoint1[19002] = {X 191.2423, Y 20.8879, Z -2.1667, A 0.000, B 0.000, C 0.000 }
gfCNCPoint1[19003] = {X 191.0007, Y 20.4545, Z -2.1667, A 0.000, B 0.000, C 0.000 }
gfCNCPoint1[19004] = {X 190.6321, Y 20.1224, Z -2.1667, A 0.000, B 0.000, C 0.000 }
gfCNCPoint1[19005] = {X 189.7428, Y 19.6452, Z -2.1667, A 0.000, B 0.000, C 0.000 }
gfCNCPoint1[19006] = {X 188.7914, Y 19.3087, Z -2.1667, A 0.000, B 0.000, C 0.000 }
gfCNCPoint1[19007] = {X 187.7998, Y 19.1206, Z -2.1667, A 0.000, B 0.000, C 0.000 }
gfCNCPoint1[19008] = {X 186.4276, Y 19.0358, Z -2.1667, A 0.000, B 0.000, C 0.000 }
gfCNCPoint1[19009] = {X 185.0543, Y 19.0995, Z -2.1667, A 0.000, B 0.000, C 0.000 }
gfCNCPoint1[19010] = {X 183.6958, Y 19.3108, Z -2.1667, A 0.000, B 0.000, C 0.000 }
gfCNCPoint1[19011] = {X 182.4009, Y 19.6817, Z -2.1667, A 0.000, B 0.000, C 0.000 }
gfCNCPoint1[19012] = {X 181.1779, Y 20.2463, Z -2.1667, A 0.000, B 0.000, C 0.000 }
gfCNCPoint1[19013] = {X 181.1606, Y 20.3407, Z -2.1667, A 0.000, B 0.000, C 0.000 }
gfCNCPoint1[19014] = {X 180.9651, Y 21.2476, Z -2.1667, A 0.000, B 0.000, C 0.000 }
gfCNCPoint1[19015] = {X 180.5735, Y 22.0886, Z -2.1667, A 0.000, B 0.000, C 0.000 }
gfCNCPoint1[19016] = {X 180.0052, Y 22.8220, Z -2.1667, A 0.000, B 0.000, C 0.000 }
gfCNCPoint1[19017] = {X 180.1927, Y 22.8279, Z -2.1667, A 0.000, B 0.000, C 0.000 }
gfCNCPoint1[19018] = {X 182.2672, Y 22.6082, Z -2.1667, A 0.000, B 0.000, C 0.000 }
gfCNCPoint1[19019] = {X 184.3489, Y 22.4744, Z -2.1667, A 0.000, B 0.000, C 0.000 }
gfCNCPoint1[19020] = {X 184.7855, Y 22.4584, Z -2.1667, A 0.000, B 0.000, C 0.000 }
gfCNCPoint1[19021] = {X 185.2220, Y 22.4408, Z -2.1667, A 0.000, B 0.000, C 0.000 }
gfCNCPoint1[19022] = {X 189.1885, Y 21.9243, Z -2.1667, A 0.000, B 0.000, C 0.000 }
gfCNCPoint1[19023] = {X 181.2295, Y 22.3407, Z -2.1667, A 0.000, B 0.000, C 0.000 }
gfCNCPoint1[19024] = {X 185.2254, Y 22.5208, Z -2.1667, A 0.000, B 0.000, C 0.000 }
gfCNCPoint1[19025] = {X 187.5588, Y 22.3980, Z -2.1667, A 0.000, B 0.000, C 0.000 }
gfCNCPoint1[19026] = {X 189.8892, Y 22.2271, Z -2.1667, A 0.000, B 0.000, C 0.000 }
gfCNCPoint1[19027] = {X 190.6154, Y 22.1295, Z -2.1667, A 0.000, B 0.000, C 0.000 }
gfCNCPoint1[19028] = {X 191.3201, Y 21.9289, Z -2.1667, A 0.000, B 0.000, C 0.000 }
gfCNCPoint1[19029] = {X 191.4109, Y 21.4046, Z -2.1667, A 0.000, B 0.000, C 0.000 }
gfCNCPoint1[19030] = {X 191.3241, Y 20.8796, Z -2.1667, A 0.000, B 0.000, C 0.000 }
gfCNCPoint1[19031] = {X 191.0694, Y 20.4124, Z -2.1667, A 0.000, B 0.000, C 0.000 }
gfCNCPoint1[19032] = {X 190.6752, Y 20.0550, Z -2.1667, A 0.000, B 0.000, C 0.000 }
gfCNCPoint1[19033] = {X 189.7752, Y 19.5720, Z -2.1667, A 0.000, B 0.000, C 0.000 }
gfCNCPoint1[19034] = {X 188.8122, Y 19.2314, Z -2.1667, A 0.000, B 0.000, C 0.000 }
gfCNCPoint1[19035] = {X 187.8087, Y 19.0411, Z -2.1667, A 0.000, B 0.000, C 0.000 }
gfCNCPoint1[19036] = {X 186.4280, Y 18.9558, Z -2.1667, A 0.000, B 0.000, C 0.000 }
gfCNCPoint1[19037] = {X 185.0461, Y 19.0199, Z -2.1667, A 0.000, B 0.000, C 0.000 }
gfCNCPoint1[19038] = {X 183.6792, Y 19.2325, Z -2.1667, A 0.000, B 0.000, C 0.000 }
gfCNCPoint1[19039] = {X 182.3551, Y 19.6134, Z -2.1667, A 0.000, B 0.000, C 0.000 }
gfCNCPoint1[19040] = {X 181.1060, Y 20.1949, Z -2.1667, A 0.000, B 0.000, C 0.000 }
gfCNCPoint1[19041] = {X 181.0813, Y 20.3295, Z -2.1667, A 0.000, B 0.000, C 0.000 }
gfCNCPoint1[19042] = {X 180.8699, Y 21.2784, Z -2.1667, A 0.000, B 0.000, C 0.000 }
gfCNCPoint1[19043] = {X 180.4399, Y 22.1505, Z -2.1667, A 0.000, B 0.000, C 0.000 }
gfCNCPoint1[19044] = {X 179.8159, Y 22.8960, Z -2.1667, A 0.000, B 0.000, C 0.000 }
gfCNCPoint1[19045] = {X 180.1965, Y 22.9081, Z -2.1667, A 0.000, B 0.000, C 0.000 }
gfCNCPoint1[19046] = {X 182.2706, Y 22.6882, Z -2.1667, A 0.000, B 0.000, C 0.000 }
gfCNCPoint1[19047] = {X 184.3521, Y 22.5543, Z -2.1667, A 0.000, B 0.000, C 0.000 }
gfCNCPoint1[19048] = {X 184.7888, Y 22.5384, Z -2.1667, A 0.000, B 0.000, C 0.000 }
gfCNCPoint1[19049] = {X 185.2254, Y 22.5208, Z -2.1667, A 0.000, B 0.000, C 0.000 }
gfCNCPoint1[19050] = {X 189.1919, Y 22.0042, Z -2.1667, A 0.000, B 0.000, C 0.000 }
gfCNCPoint1[19051] = {X 185.1537, Y 22.6038, Z -2.1667, A 0.000, B 0.000, C 0.000 }
gfCNCPoint1[19052] = {X 185.2288, Y 22.6007, Z -2.1667, A 0.000, B 0.000, C 0.000 }
gfCNCPoint1[19053] = {X 187.5634, Y 22.4779, Z -2.1667, A 0.000, B 0.000, C 0.000 }
gfCNCPoint1[19054] = {X 189.8950, Y 22.3069, Z -2.1667, A 0.000, B 0.000, C 0.000 }
gfCNCPoint1[19055] = {X 190.6504, Y 22.2039, Z -2.1667, A 0.000, B 0.000, C 0.000 }
gfCNCPoint1[19056] = {X 191.3825, Y 21.9911, Z -2.1667, A 0.000, B 0.000, C 0.000 }
gfCNCPoint1[19057] = {X 191.4906, Y 21.4333, Z -2.1667, A 0.000, B 0.000, C 0.000 }
gfCNCPoint1[19058] = {X 191.4059, Y 20.8715, Z -2.1667, A 0.000, B 0.000, C 0.000 }
gfCNCPoint1[19059] = {X 191.1381, Y 20.3704, Z -2.1667, A 0.000, B 0.000, C 0.000 }
gfCNCPoint1[19060] = {X 190.7183, Y 19.9876, Z -2.1667, A 0.000, B 0.000, C 0.000 }
gfCNCPoint1[19061] = {X 189.8075, Y 19.4989, Z -2.1667, A 0.000, B 0.000, C 0.000 }
gfCNCPoint1[19062] = {X 188.8331, Y 19.1542, Z -2.1667, A 0.000, B 0.000, C 0.000 }
gfCNCPoint1[19063] = {X 187.8176, Y 18.9616, Z -2.1667, A 0.000, B 0.000, C 0.000 }
gfCNCPoint1[19064] = {X 186.4284, Y 18.8758, Z -2.1667, A 0.000, B 0.000, C 0.000 }
gfCNCPoint1[19065] = {X 185.0380, Y 18.9403, Z -2.1667, A 0.000, B 0.000, C 0.000 }
gfCNCPoint1[19066] = {X 183.6627, Y 19.1543, Z -2.1667, A 0.000, B 0.000, C 0.000 }
gfCNCPoint1[19067] = {X 182.3093, Y 19.5452, Z -2.1667, A 0.000, B 0.000, C 0.000 }
gfCNCPoint1[19068] = {X 181.0340, Y 20.1438, Z -2.1667, A 0.000, B 0.000, C 0.000 }
gfCNCPoint1[19069] = {X 181.0020, Y 20.3183, Z -2.1667, A 0.000, B 0.000, C 0.000 }
gfCNCPoint1[19070] = {X 180.8538, Y 21.0695, Z -2.1667, A 0.000, B 0.000, C 0.000 }
gfCNCPoint1[19071] = {X 180.5651, Y 21.7787, Z -2.1667, A 0.000, B 0.000, C 0.000 }
gfCNCPoint1[19072] = {X 180.1466, Y 22.4199, Z -2.1667, A 0.000, B 0.000, C 0.000 }
gfCNCPoint1[19073] = {X 179.6136, Y 22.9696, Z -2.1667, A 0.000, B 0.000, C 0.000 }
gfCNCPoint1[19074] = {X 180.2003, Y 22.9883, Z -2.1667, A 0.000, B 0.000, C 0.000 }
gfCNCPoint1[19075] = {X 182.2741, Y 22.7682, Z -2.1667, A 0.000, B 0.000, C 0.000 }
gfCNCPoint1[19076] = {X 184.3552, Y 22.6342, Z -2.1667, A 0.000, B 0.000, C 0.000 }
gfCNCPoint1[19077] = {X 184.7920, Y 22.6183, Z -2.1667, A 0.000, B 0.000, C 0.000 }
gfCNCPoint1[19078] = {X 185.2288, Y 22.6007, Z -2.1667, A 0.000, B 0.000, C 0.000 }
gfCNCPoint1[19079] = {X 185.1443, Y 20.6025, Z -2.1667, A 0.000, B 0.000, C 0.000 }
gfCNCPoint1[19080] = {X 185.1443, Y 20.6025, Z 0.8333, A 0.000, B 0.000, C 0.000 }
gfCNCPoint1[19081] = {X 185.1443, Y 20.6025, Z 11.0000, A 0.000, B 0.000, C 0.000 }
gfCNCPoint1[19082] = {X 256.2418, Y 19.7801, Z 11.0000, A 0.000, B 0.000, C 0.000 }
gfCNCPoint1[19083] = {X 256.2418, Y 19.7801, Z 1.6667, A 0.000, B 0.000, C 0.000 }
gfCNCPoint1[19084] = {X 251.5292, Y 19.7801, Z 0.4039, A 0.000, B 0.000, C 0.000 }
gfCNCPoint1[19085] = {X 250.8346, Y 19.7909, Z 0.2178, A 0.000, B 0.000, C 0.000 }
gfCNCPoint1[19086] = {X 250.1804, Y 19.7926, Z 0.0425, A 0.000, B 0.000, C 0.000 }
gfCNCPoint1[19087] = {X 249.4960, Y 19.8908, Z -0.1428, A 0.000, B 0.000, C 0.000 }
gfCNCPoint1[19088] = {X 248.8451, Y 20.0790, Z -0.3243, A 0.000, B 0.000, C 0.000 }
gfCNCPoint1[19089] = {X 248.7080, Y 20.1103, Z -0.3620, A 0.000, B 0.000, C 0.000 }
gfCNCPoint1[19090] = {X 248.6534, Y 20.1615, Z -0.3820, A 0.000, B 0.000, C 0.000 }
gfCNCPoint1[19091] = {X 248.6134, Y 20.2963, Z -0.4197, A 0.000, B 0.000, C 0.000 }
gfCNCPoint1[19092] = {X 248.4743, Y 20.7644, Z -0.5506, A 0.000, B 0.000, C 0.000 }
gfCNCPoint1[19093] = {X 248.4443, Y 21.8682, Z -0.8465, A 0.000, B 0.000, C 0.000 }
gfCNCPoint1[19094] = {X 248.5576, Y 22.3432, Z -0.9773, A 0.000, B 0.000, C 0.000 }
gfCNCPoint1[19095] = {X 248.8713, Y 22.4375, Z -1.0651, A 0.000, B 0.000, C 0.000 }
gfCNCPoint1[19096] = {X 249.1976, Y 22.4648, Z -1.1528, A 0.000, B 0.000, C 0.000 }
gfCNCPoint1[19097] = {X 250.4383, Y 22.5687, Z -1.4864, A 0.000, B 0.000, C 0.000 }
gfCNCPoint1[19098] = {X 251.6873, Y 22.5560, Z -1.8211, A 0.000, B 0.000, C 0.000 }
gfCNCPoint1[19099] = {X 252.9770, Y 22.5560, Z -2.1667, A 0.000, B 0.000, C 0.000 }
gfCNCPoint1[19100] = {X 257.4115, Y 22.5560, Z -2.1667, A 0.000, B 0.000, C 0.000 }
gfCNCPoint1[19101] = {X 257.4115, Y 19.7801, Z -2.1667, A 0.000, B 0.000, C 0.000 }
gfCNCPoint1[19102] = {X 251.5292, Y 19.7801, Z -2.1667, A 0.000, B 0.000, C 0.000 }
gfCNCPoint1[19103] = {X 250.8346, Y 19.7909, Z -2.1667, A 0.000, B 0.000, C 0.000 }
gfCNCPoint1[19104] = {X 249.8297, Y 19.8644, Z -2.1667, A 0.000, B 0.000, C 0.000 }
gfCNCPoint1[19105] = {X 248.8451, Y 20.0790, Z -2.1667, A 0.000, B 0.000, C 0.000 }
gfCNCPoint1[19106] = {X 248.6998, Y 20.1563, Z -2.1667, A 0.000, B 0.000, C 0.000 }
gfCNCPoint1[19107] = {X 248.6134, Y 20.2963, Z -2.1667, A 0.000, B 0.000, C 0.000 }
gfCNCPoint1[19108] = {X 248.4753, Y 20.9719, Z -2.1667, A 0.000, B 0.000, C 0.000 }
gfCNCPoint1[19109] = {X 248.4566, Y 21.6612, Z -2.1667, A 0.000, B 0.000, C 0.000 }
gfCNCPoint1[19110] = {X 248.5576, Y 22.3432, Z -2.1667, A 0.000, B 0.000, C 0.000 }
gfCNCPoint1[19111] = {X 248.8745, Y 22.4207, Z -2.1667, A 0.000, B 0.000, C 0.000 }
gfCNCPoint1[19112] = {X 249.1976, Y 22.4648, Z -2.1667, A 0.000, B 0.000, C 0.000 }
gfCNCPoint1[19113] = {X 250.4414, Y 22.5397, Z -2.1667, A 0.000, B 0.000, C 0.000 }
gfCNCPoint1[19114] = {X 251.6873, Y 22.5560, Z -2.1667, A 0.000, B 0.000, C 0.000 }
gfCNCPoint1[19115] = {X 252.9770, Y 22.5560, Z -2.1667, A 0.000, B 0.000, C 0.000 }
gfCNCPoint1[19116] = {X 248.9922, Y 22.2874, Z -2.1667, A 0.000, B 0.000, C 0.000 }
gfCNCPoint1[19117] = {X 252.9770, Y 22.6360, Z -2.1667, A 0.000, B 0.000, C 0.000 }
gfCNCPoint1[19118] = {X 257.4915, Y 22.6360, Z -2.1667, A 0.000, B 0.000, C 0.000 }
gfCNCPoint1[19119] = {X 257.4915, Y 19.7001, Z -2.1667, A 0.000, B 0.000, C 0.000 }
gfCNCPoint1[19120] = {X 251.5286, Y 19.7001, Z -2.1667, A 0.000, B 0.000, C 0.000 }
gfCNCPoint1[19121] = {X 250.8365, Y 19.7109, Z -2.1667, A 0.000, B 0.000, C 0.000 }
gfCNCPoint1[19122] = {X 249.8259, Y 19.7845, Z -2.1667, A 0.000, B 0.000, C 0.000 }
gfCNCPoint1[19123] = {X 248.8355, Y 19.9992, Z -2.1667, A 0.000, B 0.000, C 0.000 }
gfCNCPoint1[19124] = {X 248.6482, Y 20.0951, Z -2.1667, A 0.000, B 0.000, C 0.000 }
gfCNCPoint1[19125] = {X 248.5367, Y 20.2735, Z -2.1667, A 0.000, B 0.000, C 0.000 }
gfCNCPoint1[19126] = {X 248.3941, Y 20.9779, Z -2.1667, A 0.000, B 0.000, C 0.000 }
gfCNCPoint1[19127] = {X 248.3786, Y 21.6964, Z -2.1667, A 0.000, B 0.000, C 0.000 }
gfCNCPoint1[19128] = {X 248.4907, Y 22.4063, Z -2.1667, A 0.000, B 0.000, C 0.000 }
gfCNCPoint1[19129] = {X 248.8370, Y 22.4949, Z -2.1667, A 0.000, B 0.000, C 0.000 }
gfCNCPoint1[19130] = {X 249.1909, Y 22.5446, Z -2.1667, A 0.000, B 0.000, C 0.000 }
gfCNCPoint1[19131] = {X 250.4372, Y 22.6196, Z -2.1667, A 0.000, B 0.000, C 0.000 }
gfCNCPoint1[19132] = {X 251.6857, Y 22.6360, Z -2.1667, A 0.000, B 0.000, C 0.000 }
gfCNCPoint1[19133] = {X 252.9770, Y 22.6360, Z -2.1667, A 0.000, B 0.000, C 0.000 }
gfCNCPoint1[19134] = {X 256.9618, Y 22.2874, Z -2.1667, A 0.000, B 0.000, C 0.000 }
gfCNCPoint1[19135] = {X 248.9922, Y 22.3674, Z -2.1667, A 0.000, B 0.000, C 0.000 }
gfCNCPoint1[19136] = {X 252.9770, Y 22.7160, Z -2.1667, A 0.000, B 0.000, C 0.000 }
gfCNCPoint1[19137] = {X 257.5715, Y 22.7160, Z -2.1667, A 0.000, B 0.000, C 0.000 }
gfCNCPoint1[19138] = {X 257.5715, Y 19.6201, Z -2.1667, A 0.000, B 0.000, C 0.000 }
gfCNCPoint1[19139] = {X 251.5280, Y 19.6201, Z -2.1667, A 0.000, B 0.000, C 0.000 }
gfCNCPoint1[19140] = {X 250.8358, Y 19.6309, Z -2.1667, A 0.000, B 0.000, C 0.000 }
gfCNCPoint1[19141] = {X 249.8156, Y 19.7051, Z -2.1667, A 0.000, B 0.000, C 0.000 }
gfCNCPoint1[19142] = {X 248.8160, Y 19.9216, Z -2.1667, A 0.000, B 0.000, C 0.000 }
gfCNCPoint1[19143] = {X 248.5928, Y 20.0373, Z -2.1667, A 0.000, B 0.000, C 0.000 }
gfCNCPoint1[19144] = {X 248.4600, Y 20.2508, Z -2.1667, A 0.000, B 0.000, C 0.000 }
gfCNCPoint1[19145] = {X 248.3130, Y 20.9838, Z -2.1667, A 0.000, B 0.000, C 0.000 }
gfCNCPoint1[19146] = {X 248.3009, Y 21.7314, Z -2.1667, A 0.000, B 0.000, C 0.000 }
gfCNCPoint1[19147] = {X 248.4242, Y 22.4688, Z -2.1667, A 0.000, B 0.000, C 0.000 }
gfCNCPoint1[19148] = {X 248.7996, Y 22.5690, Z -2.1667, A 0.000, B 0.000, C 0.000 }
gfCNCPoint1[19149] = {X 249.1842, Y 22.6243, Z -2.1667, A 0.000, B 0.000, C 0.000 }
gfCNCPoint1[19150] = {X 250.4341, Y 22.6995, Z -2.1667, A 0.000, B 0.000, C 0.000 }
gfCNCPoint1[19151] = {X 251.6861, Y 22.7160, Z -2.1667, A 0.000, B 0.000, C 0.000 }
gfCNCPoint1[19152] = {X 252.9770, Y 22.7160, Z -2.1667, A 0.000, B 0.000, C 0.000 }
gfCNCPoint1[19153] = {X 256.9618, Y 22.3674, Z -2.1667, A 0.000, B 0.000, C 0.000 }
gfCNCPoint1[19154] = {X 248.9922, Y 22.4474, Z -2.1667, A 0.000, B 0.000, C 0.000 }
gfCNCPoint1[19155] = {X 252.9770, Y 22.7960, Z -2.1667, A 0.000, B 0.000, C 0.000 }
gfCNCPoint1[19156] = {X 257.6515, Y 22.7960, Z -2.1667, A 0.000, B 0.000, C 0.000 }
gfCNCPoint1[19157] = {X 257.6515, Y 19.5401, Z -2.1667, A 0.000, B 0.000, C 0.000 }
gfCNCPoint1[19158] = {X 251.5274, Y 19.5401, Z -2.1667, A 0.000, B 0.000, C 0.000 }
gfCNCPoint1[19159] = {X 250.8351, Y 19.5509, Z -2.1667, A 0.000, B 0.000, C 0.000 }
gfCNCPoint1[19160] = {X 249.8053, Y 19.6258, Z -2.1667, A 0.000, B 0.000, C 0.000 }
gfCNCPoint1[19161] = {X 248.7962, Y 19.8441, Z -2.1667, A 0.000, B 0.000, C 0.000 }
gfCNCPoint1[19162] = {X 248.5373, Y 19.9797, Z -2.1667, A 0.000, B 0.000, C 0.000 }
gfCNCPoint1[19163] = {X 248.3833, Y 20.2280, Z -2.1667, A 0.000, B 0.000, C 0.000 }
gfCNCPoint1[19164] = {X 248.2320, Y 20.9896, Z -2.1667, A 0.000, B 0.000, C 0.000 }
gfCNCPoint1[19165] = {X 248.2234, Y 21.7661, Z -2.1667, A 0.000, B 0.000, C 0.000 }
gfCNCPoint1[19166] = {X 248.3580, Y 22.5309, Z -2.1667, A 0.000, B 0.000, C 0.000 }
gfCNCPoint1[19167] = {X 248.7624, Y 22.6430, Z -2.1667, A 0.000, B 0.000, C 0.000 }
gfCNCPoint1[19168] = {X 249.1776, Y 22.7040, Z -2.1667, A 0.000, B 0.000, C 0.000 }
gfCNCPoint1[19169] = {X 250.4310, Y 22.7794, Z -2.1667, A 0.000, B 0.000, C 0.000 }
gfCNCPoint1[19170] = {X 251.6865, Y 22.7960, Z -2.1667, A 0.000, B 0.000, C 0.000 }
gfCNCPoint1[19171] = {X 252.9770, Y 22.7960, Z -2.1667, A 0.000, B 0.000, C 0.000 }
gfCNCPoint1[19172] = {X 256.9618, Y 22.4474, Z -2.1667, A 0.000, B 0.000, C 0.000 }
gfCNCPoint1[19173] = {X 248.9922, Y 22.5274, Z -2.1667, A 0.000, B 0.000, C 0.000 }
gfCNCPoint1[19174] = {X 252.9770, Y 22.8760, Z -2.1667, A 0.000, B 0.000, C 0.000 }
gfCNCPoint1[19175] = {X 257.7315, Y 22.8760, Z -2.1667, A 0.000, B 0.000, C 0.000 }
gfCNCPoint1[19176] = {X 257.7315, Y 19.4601, Z -2.1667, A 0.000, B 0.000, C 0.000 }
gfCNCPoint1[19177] = {X 251.5267, Y 19.4601, Z -2.1667, A 0.000, B 0.000, C 0.000 }
gfCNCPoint1[19178] = {X 250.8344, Y 19.4709, Z -2.1667, A 0.000, B 0.000, C 0.000 }
gfCNCPoint1[19179] = {X 249.7949, Y 19.5465, Z -2.1667, A 0.000, B 0.000, C 0.000 }
gfCNCPoint1[19180] = {X 248.7763, Y 19.7665, Z -2.1667, A 0.000, B 0.000, C 0.000 }
gfCNCPoint1[19181] = {X 248.4818, Y 19.9220, Z -2.1667, A 0.000, B 0.000, C 0.000 }
gfCNCPoint1[19182] = {X 248.3066, Y 20.2052, Z -2.1667, A 0.000, B 0.000, C 0.000 }
gfCNCPoint1[19183] = {X 248.1516, Y 20.9889, Z -2.1667, A 0.000, B 0.000, C 0.000 }
gfCNCPoint1[19184] = {X 248.1449, Y 21.7877, Z -2.1667, A 0.000, B 0.000, C 0.000 }
gfCNCPoint1[19185] = {X 248.2868, Y 22.5739, Z -2.1667, A 0.000, B 0.000, C 0.000 }
gfCNCPoint1[19186] = {X 248.3055, Y 22.5973, Z -2.1667, A 0.000, B 0.000, C 0.000 }
gfCNCPoint1[19187] = {X 248.3318, Y 22.6065, Z -2.1667, A 0.000, B 0.000, C 0.000 }
gfCNCPoint1[19188] = {X 248.7458, Y 22.7213, Z -2.1667, A 0.000, B 0.000, C 0.000 }
gfCNCPoint1[19189] = {X 249.1709, Y 22.7837, Z -2.1667, A 0.000, B 0.000, C 0.000 }
gfCNCPoint1[19190] = {X 250.4278, Y 22.8594, Z -2.1667, A 0.000, B 0.000, C 0.000 }
gfCNCPoint1[19191] = {X 251.6869, Y 22.8760, Z -2.1667, A 0.000, B 0.000, C 0.000 }
gfCNCPoint1[19192] = {X 252.9770, Y 22.8760, Z -2.1667, A 0.000, B 0.000, C 0.000 }
gfCNCPoint1[19193] = {X 256.9618, Y 22.5274, Z -2.1667, A 0.000, B 0.000, C 0.000 }
gfCNCPoint1[19194] = {X 248.9922, Y 22.6074, Z -2.1667, A 0.000, B 0.000, C 0.000 }
gfCNCPoint1[19195] = {X 252.9770, Y 22.9560, Z -2.1667, A 0.000, B 0.000, C 0.000 }
gfCNCPoint1[19196] = {X 257.8115, Y 22.9560, Z -2.1667, A 0.000, B 0.000, C 0.000 }
gfCNCPoint1[19197] = {X 257.8098, Y 19.3801, Z -2.1667, A 0.000, B 0.000, C 0.000 }
gfCNCPoint1[19198] = {X 251.5261, Y 19.3801, Z -2.1667, A 0.000, B 0.000, C 0.000 }
gfCNCPoint1[19199] = {X 250.8336, Y 19.3909, Z -2.1667, A 0.000, B 0.000, C 0.000 }
gfCNCPoint1[19200] = {X 249.7845, Y 19.4671, Z -2.1667, A 0.000, B 0.000, C 0.000 }
gfCNCPoint1[19201] = {X 248.7562, Y 19.6891, Z -2.1667, A 0.000, B 0.000, C 0.000 }
gfCNCPoint1[19202] = {X 248.4263, Y 19.8645, Z -2.1667, A 0.000, B 0.000, C 0.000 }
gfCNCPoint1[19203] = {X 248.2299, Y 20.1824, Z -2.1667, A 0.000, B 0.000, C 0.000 }
gfCNCPoint1[19204] = {X 248.0715, Y 20.9862, Z -2.1667, A 0.000, B 0.000, C 0.000 }
gfCNCPoint1[19205] = {X 248.0662, Y 21.8054, Z -2.1667, A 0.000, B 0.000, C 0.000 }
gfCNCPoint1[19206] = {X 248.2142, Y 22.6111, Z -2.1667, A 0.000, B 0.000, C 0.000 }
gfCNCPoint1[19207] = {X 248.2572, Y 22.6650, Z -2.1667, A 0.000, B 0.000, C 0.000 }
gfCNCPoint1[19208] = {X 248.7041, Y 22.7941, Z -2.1667, A 0.000, B 0.000, C 0.000 }
gfCNCPoint1[19209] = {X 249.1642, Y 22.8634, Z -2.1667, A 0.000, B 0.000, C 0.000 }
gfCNCPoint1[19210] = {X 250.4247, Y 22.9393, Z -2.1667, A 0.000, B 0.000, C 0.000 }
gfCNCPoint1[19211] = {X 251.6873, Y 22.9560, Z -2.1667, A 0.000, B 0.000, C 0.000 }
gfCNCPoint1[19212] = {X 252.9770, Y 22.9560, Z -2.1667, A 0.000, B 0.000, C 0.000 }
gfCNCPoint1[19213] = {X 256.9618, Y 22.6074, Z -2.1667, A 0.000, B 0.000, C 0.000 }
gfCNCPoint1[19214] = {X 256.9618, Y 22.6074, Z 0.8333, A 0.000, B 0.000, C 0.000 }
gfCNCPoint1[19215] = {X 256.9618, Y 22.6074, Z 11.0000, A 0.000, B 0.000, C 0.000 }
gfCNCPoint1[19216] = {X 507.6819, Y 107.6949, Z 11.0000, A 0.000, B 0.000, C 0.000 }
gfCNCPoint1[19217] = {X 507.6819, Y 107.6949, Z 0.8333, A 0.000, B 0.000, C 0.000 }
gfCNCPoint1[19218] = {X 507.6819, Y 107.6949, Z -2.1667, A 0.000, B 0.000, C 0.000 }
gfCNCPoint1[19219] = {X 507.6819, Y 71.2949, Z -2.1667, A 0.000, B 0.000, C 0.000 }
gfCNCPoint1[19220] = {X 509.5499, Y 71.2949, Z -2.1667, A 0.000, B 0.000, C 0.000 }
gfCNCPoint1[19221] = {X 509.0277, Y 71.0691, Z -2.1667, A 0.000, B 0.000, C 0.000 }
gfCNCPoint1[19222] = {X 508.5105, Y 70.8320, Z -2.1667, A 0.000, B 0.000, C 0.000 }
gfCNCPoint1[19223] = {X 507.1681, Y 71.0983, Z -2.1667, A 0.000, B 0.000, C 0.000 }
gfCNCPoint1[19224] = {X 505.8138, Y 71.2949, Z -2.1667, A 0.000, B 0.000, C 0.000 }
gfCNCPoint1[19225] = {X 507.6819, Y 71.2949, Z -2.1667, A 0.000, B 0.000, C 0.000 }
gfCNCPoint1[19226] = {X 507.6819, Y 73.6949, Z -2.1667, A 0.000, B 0.000, C 0.000 }
gfCNCPoint1[19227] = {X 551.2532, Y 73.6949, Z -2.1667, A 0.000, B 0.000, C 0.000 }
gfCNCPoint1[19228] = {X 549.1233, Y 72.7703, Z -2.1667, A 0.000, B 0.000, C 0.000 }
gfCNCPoint1[19229] = {X 547.0690, Y 71.6879, Z -2.1667, A 0.000, B 0.000, C 0.000 }
gfCNCPoint1[19230] = {X 545.1022, Y 70.4537, Z -2.1667, A 0.000, B 0.000, C 0.000 }
gfCNCPoint1[19231] = {X 543.2340, Y 69.0749, Z -2.1667, A 0.000, B 0.000, C 0.000 }
gfCNCPoint1[19232] = {X 529.7641, Y 69.0753, Z -2.1667, A 0.000, B 0.000, C 0.000 }
gfCNCPoint1[19233] = {X 527.5535, Y 69.8782, Z -2.1667, A 0.000, B 0.000, C 0.000 }
gfCNCPoint1[19234] = {X 525.2755, Y 70.4630, Z -2.1667, A 0.000, B 0.000, C 0.000 }
gfCNCPoint1[19235] = {X 522.9516, Y 70.8244, Z -2.1667, A 0.000, B 0.000, C 0.000 }
gfCNCPoint1[19236] = {X 520.6036, Y 70.9588, Z -2.1667, A 0.000, B 0.000, C 0.000 }
